// TIA Portal project "997CS100_KKD" (V16)

(* hardware
DEVICE "S71500/ET200MP station_1"  S7-1500 station
   slot 0: "-N01.01.00"  Rack  6ES7 590-1***0-0AA0
   slot 1: "997CS100"  CPU 1515-2 PN  6ES7 515-2AM02-0AB0  V2.8
      slot 3: "CPU display_1"  6ES7591-1BA00-0AA0
      slot 32768: "IO"  X1
      slot 33024: "PROFINET interface_1"  X2
      slot 34817: "Virtual CP interface port_1"  Virtual CP interface port  Virtual CP interface port
DEVICE "Station ET 200SP_7"  ET 200SP-Station
   slot 0: "Châssis_0"  6ES5 710-8MAx1
   slot 0: "PMC"  IM 155-6 PN ST  6ES7 155-6AU01-0BN0  V4.1
   slot 1: "501DI1"  DI 16x24VDC ST  6ES7 131-6BH01-0BA0  V0.0
      slot 1: "501DI1"  DI 16x24VDC ST
   slot 2: "501DI2"  DI 16x24VDC ST  6ES7 131-6BH01-0BA0  V0.0
      slot 1: "501DI2"  DI 16x24VDC ST
   slot 3: "501DI3"  DI 16x24VDC ST  6ES7 131-6BH01-0BA0  V0.0
      slot 1: "501DI3"  DI 16x24VDC ST
   slot 4: "501DI4"  DI 16x24VDC ST  6ES7 131-6BH01-0BA0  V0.0
      slot 1: "501DI4"  DI 16x24VDC ST
   slot 5: "501DI5"  DI 16x24VDC ST  6ES7 131-6BH01-0BA0  V0.0
      slot 1: "501DI5"  DI 16x24VDC ST
   slot 6: "502DO1"  RQ 4x120VDC/230VAC/5A NO ST  6ES7 132-6HD01-0BB1  V0.0
      slot 1: "502DO1"  RQ 4x120VDC/230VAC/5A NO ST
   slot 7: "502DO2"  RQ 4x120VDC/230VAC/5A NO ST  6ES7 132-6HD01-0BB1  V0.0
      slot 1: "502DO2"  RQ 4x120VDC/230VAC/5A NO ST
   slot 8: "502DO3"  RQ 4x120VDC/230VAC/5A NO ST  6ES7 132-6HD01-0BB1  V0.0
      slot 1: "502DO3"  RQ 4x120VDC/230VAC/5A NO ST
   slot 9: "502DO4"  RQ 4x120VDC/230VAC/5A NO ST  6ES7 132-6HD01-0BB1  V0.0
      slot 1: "502DO4"  RQ 4x120VDC/230VAC/5A NO ST
   slot 10: "502AI1"  AI 4xI 2-,4-wire ST  6ES7 134-6GD01-0BA1  V2.0
      slot 1: "502AI1"  AI 4xI 2-,4-wire ST
   slot 11: "502AI2"  AI 4xI 2-,4-wire ST  6ES7 134-6GD01-0BA1  V2.0
      slot 1: "502AI2"  AI 4xI 2-,4-wire ST
   slot 12: "502AI3"  AI 8xI 2-,4-wire BA  6ES7 134-6GF00-0AA1  V1.0
      slot 1: "502AI3"  AI 8xI 2-,4-wire BA
   slot 13: "300DI1"  DI 16x24VDC ST  6ES7 131-6BH01-0BA0  V0.0
      slot 1: "300DI1"  DI 16x24VDC ST
   slot 14: "300DI2"  DI 16x24VDC ST  6ES7 131-6BH01-0BA0  V0.0
      slot 1: "300DI2"  DI 16x24VDC ST
   slot 15: "300DI3"  DI 16x24VDC ST  6ES7 131-6BH01-0BA0  V0.0
      slot 1: "300DI3"  DI 16x24VDC ST
   slot 16: "300DO1"  DQ 16x24VDC/0.5A ST  6ES7 132-6BH01-0BA0  V0.0
      slot 1: "300DO1"  DQ 16x24VDC/0.5A ST
   slot 17: "Module serveur_1"  Module serveur  6ES7 193-6PA00-0AA0  V1.0
      slot 1: "Module serveur_1"  Module serveur
   slot 127: "Adaptateur de bus PROFINET CU"  PROFINET Interface  6ES7 193-6AR00-0AA0  V0.0
      slot 1: "Port_1"  6ES7 193-6AR00-0AA0  V0.0
      slot 2: "Port_2"  6ES7 193-6AR00-0AA0  V0.0
DEVICE "GSD device_2"  GSD.Device.PN
   slot 0: "Rack"  Rack  V1.0
   slot 0: "CV180_VFD"  INVT Profinet Adapter V1.0  1234567  V13.00.00
      slot 0: "INVT Profinet Adapter board V1.0"  INVT Profinet Adapter board V1.0
      slot 1: "PN-IO"  PN-IO
         slot 1: "Port 1 - RJ45"  Port 1 - RJ45
         slot 2: "Port 2 - RJ45"  Port 2 - RJ45
   slot 1: "32 Byte IN/OUT_1"  32 Byte IN/OUT  1.0
      slot 0: "32 Byte IN/OUT"  32 Byte IN/OUT
DEVICE "2010CV300U01_INVT"  GSD.Device.PN
   slot 0: "Rack"  Rack  V1.0
   slot 0: "2010CV300U01_INVT"  INVT Profinet Adapter V1.0  1234567  V13.00.00
      slot 0: "INVT Profinet Adapter board V1.0"  INVT Profinet Adapter board V1.0
      slot 1: "PN-IO"  PN-IO
         slot 1: "Port 1 - RJ45"  Port 1 - RJ45
         slot 2: "Port 2 - RJ45"  Port 2 - RJ45
   slot 1: "32 Byte IN/OUT_1"  32 Byte IN/OUT  1.0
      slot 0: "32 Byte IN/OUT"  32 Byte IN/OUT
DEVICE "Control device Station"  SIMOCODE pro
   slot 0: "Rack"  Rail
   slot 0: "2010cv120m01"  SIMOCODE pro V PN  3UF7 011-1A*00-0  V2.1
      slot 1: "Control device IO_1"  3UF7 011-1A*00-0
   slot 101: "IM 2.4 - 25A"  Current measuring module 2.4..25A  3UF7 101-1*A00-0
DEVICE "ET 200SP station_1"  ET 200SP-Station
   slot 0: "-N02.01.00"  Rack  6ES5 710-8MAx1
   slot 0: "993CS110A01"  IM 155-6 PN/2 HF  6ES7 155-6AU01-0CN0  V4.2
   slot 1: "-N02.01.01"  DI 16x24VDC ST  6ES7 131-6BH01-0BA0  V0.0
      slot 1: "-N02.01.01"  DI 16x24VDC ST
   slot 2: "-N02.01.02"  AI 8xI 2-,4-wire BA  6ES7 134-6GF00-0AA1  V1.0
      slot 1: "-N02.01.02"  AI 8xI 2-,4-wire BA
   slot 3: "-N02.01.03"  AQ 4xU/I ST  6ES7 135-6HD00-0BA1  V1.1
      slot 1: "-N02.01.03"  AQ 4xU/I ST
   slot 4: "-N02.01.04"  DI 16x24VDC ST  6ES7 131-6BH01-0BA0  V0.0
      slot 1: "-N02.01.04"  DI 16x24VDC ST
   slot 5: "-N02.01.05"  DI 16x24VDC ST  6ES7 131-6BH01-0BA0  V0.0
      slot 1: "-N02.01.05"  DI 16x24VDC ST
   slot 6: "-N02.01.06"  DI 16x24VDC ST  6ES7 131-6BH01-0BA0  V0.0
      slot 1: "-N02.01.06"  DI 16x24VDC ST
   slot 7: "-N02.01.07"  DQ 16x24VDC/0.5A ST  6ES7 132-6BH01-0BA0  V0.0
      slot 1: "-N02.01.07"  DQ 16x24VDC/0.5A ST
   slot 8: "-N02.01.08"  DQ 16x24VDC/0.5A ST  6ES7 132-6BH01-0BA0  V0.0
      slot 1: "-N02.01.08"  DQ 16x24VDC/0.5A ST
   slot 9: "-N02.01.09"  DQ 16x24VDC/0.5A ST  6ES7 132-6BH01-0BA0  V0.0
      slot 1: "-N02.01.09"  DQ 16x24VDC/0.5A ST
   slot 10: "Server module_1"  Server module  6ES7 193-6PA00-0AA0  V1.1
      slot 1: "Server module_1"  Server module
   slot 127: "BA 2xRJ45"  BA 2xRJ45  6ES7 193-6AR00-0AA0  V0.0
      slot 1: "Port_1"  X1 P1 R  6ES7 193-6AR00-0AA0  V0.0
      slot 2: "Port_2"  X1 P2 R  6ES7 193-6AR00-0AA0  V0.0
DEVICE "997spareABB1"  GSD.Device.PN
   slot 0: "Rack"  Rack  V1.0
   slot 0: "997spareABB1"  FENA-21  6438177287452  V3.2.0
      slot 0: "FENA-21"  FENA-21
      slot 1: "997spareABB1"  Interface
         slot 1: "Port 1"  Port 1
         slot 2: "Port 2"  Port 2
   slot 1: "PPO Type 7_1"  PPO Type 7  V3.2.0
      slot 0: "PPO7 Data Object"  PPO7 Data Object
DEVICE "2015PU040U01"  GSD.Device.PN
   slot 0: "Rack"  Rack  V1.0
   slot 0: "2015PU040U01"  FENA-21  6438177287452  V3.2.0
      slot 0: "FENA-21"  FENA-21
      slot 1: "Interface"  Interface
         slot 1: "Port 1"  Port 1
         slot 2: "Port 2"  Port 2
   slot 1: "PPO Type 7_1"  PPO Type 7  V3.2.0
      slot 0: "PPO7 Data Object"  PPO7 Data Object
DEVICE "2015PU027U01"  GSD.Device.PN
   slot 0: "Rack"  Rack  V1.0
   slot 0: "2015PU027U01"  INVT Profinet Adapter V1.0  1234567  V13.00.00
      slot 0: "INVT Profinet Adapter board V1.0"  INVT Profinet Adapter board V1.0
      slot 1: "PN-IO"  PN-IO
         slot 1: "Port 1 - RJ45"  Port 1 - RJ45
         slot 2: "Port 2 - RJ45"  Port 2 - RJ45
   slot 1: "32 Byte IN/OUT_1"  32 Byte IN/OUT  1.0
      slot 0: "32 Byte IN/OUT"  32 Byte IN/OUT
DEVICE "2015PU028U01"  GSD.Device.PN
   slot 0: "Rack"  Rack  V1.0
   slot 0: "2015PU028U01"  INVT Profinet Adapter V1.0  1234567  V13.00.00
      slot 0: "INVT Profinet Adapter board V1.0"  INVT Profinet Adapter board V1.0
      slot 1: "PN-IO"  PN-IO
         slot 1: "Port 1 - RJ45"  Port 1 - RJ45
         slot 2: "Port 2 - RJ45"  Port 2 - RJ45
   slot 1: "32 Byte IN/OUT_1"  32 Byte IN/OUT  1.0
      slot 0: "32 Byte IN/OUT"  32 Byte IN/OUT
DEVICE "2015PU035U01"  GSD.Device.PN
   slot 0: "Rack"  Rack  V1.0
   slot 0: "2015PU035U01"  INVT Profinet Adapter V1.0  1234567  V13.00.00
      slot 0: "INVT Profinet Adapter board V1.0"  INVT Profinet Adapter board V1.0
      slot 1: "PN-IO"  PN-IO
         slot 1: "Port 1 - RJ45"  Port 1 - RJ45
         slot 2: "Port 2 - RJ45"  Port 2 - RJ45
   slot 1: "32 Byte IN/OUT_1"  32 Byte IN/OUT  1.0
      slot 0: "32 Byte IN/OUT"  32 Byte IN/OUT
DEVICE "2015PU042M01"  SIMOCODE pro
   slot 0: "UR"  Rail
   slot 0: "2015PU042M01"  SIMOCODE pro V PN GP  3UF7 011-1A*00-1  V2.1
      slot 1: "SIMOCODE"  3UF7 011-1A*00-1
   slot 10: "OP"  Operator Panel Titangrey  3UF7 200-1AA01-0
   slot 101: "IM 10-100A"  Current measuring module 10..100A  3UF7 102-1*A00-0
DEVICE "GSD device_3"  GSD.Device.PN
   slot 0: "Rack"  Rack  V1.0
   slot 0: "BF110_VFD"  ATV930  ATV930
      slot 0: "ATV930"  ATV930
      slot 1: "Interface"  Interface
         slot 1: "Port 1"  Port 1
         slot 2: "Port 2"  Port 2
   slot 1: "Telegram 107 (4PKW/16PZD)"  Telegram 107 (4PKW/16PZD)
      slot 0: "Telegram 107"  Telegram 107
DEVICE "GSD device_4"  GSD.Device.PN
   slot 0: "Rack"  Rack  V1.0
   slot 0: "SC130_VFD"  ATV930  ATV930
      slot 0: "ATV930"  ATV930
      slot 1: "Interface"  Interface
         slot 1: "Port 1"  Port 1
         slot 2: "Port 2"  Port 2
   slot 1: "Telegram 107 (4PKW/16PZD)"  Telegram 107 (4PKW/16PZD)
      slot 0: "Telegram 107"  Telegram 107
DEVICE "2010LV100P01"  GSD.Device.PN
   slot 0: "UR"  Rack  V1.0
   slot 0: "2010LV100P01"  PAC3220
      slot 0: "PAC3220"  PAC3220
      slot 1: "2010LV100P01"  PN-IO
         slot 1: "Port 1"  Port 1
         slot 2: "Port 2"  Port 2
   slot 1: "Digital Inputs Status"  Digital Inputs Status
      slot 0: "Digital Inputs Status"  Digital Inputs Status
   slot 2: "Voltage L1-L2"  Voltage L1-L2
      slot 0: "Voltage L1-L2"  Voltage L1-L2
   slot 3: "Voltage L2-L3"  Voltage L2-L3
      slot 0: "Voltage L2-L3"  Voltage L2-L3
   slot 4: "Voltage L3-L1"  Voltage L3-L1
      slot 0: "Voltage L3-L1"  Voltage L3-L1
   slot 5: "Current L1"  Current L1
      slot 0: "Current L1"  Current L1
   slot 6: "Current L2"  Current L2
      slot 0: "Current L2"  Current L2
   slot 7: "Current L3"  Current L3
      slot 0: "Current L3"  Current L3
   slot 8: "Line Frequency"  Line Frequency
      slot 0: "Line Frequency"  Line Frequency
   slot 9: "Total Apparent Power"  Total Apparent Power
      slot 0: "Total Apparent Power"  Total Apparent Power
   slot 10: "Total Active Power"  Total Active Power
      slot 0: "Total Active Power"  Total Active Power
   slot 11: "Total Reac Power"  Total Reac Power
      slot 0: "Total Reac Power"  Total Reac Power
   slot 12: "Total Power Factor"  Total Power Factor
      slot 0: "Total Power Factor"  Total Power Factor
   slot 13: "Act Energy Imp Tar 1(F)"  Act Energy Imp Tar 1(F)
      slot 0: "Act Energy Imp Tar 1(F)"  Act Energy Imp Tar 1(F)
   slot 14: "Reac En Imp Tar 1 (F)"  Reac En Imp Tar 1 (F)
      slot 0: "Reac En Imp Tar 1 (F)"  Reac En Imp Tar 1 (F)
   slot 15: "App Energy Tariff 1 (F)"  App Energy Tariff 1 (F)
      slot 0: "App Energy Tariff 1 (F)"  App Energy Tariff 1 (F)
DEVICE "Control device Station_1"  SIMOCODE pro
   slot 0: "Rack"  Rail
   slot 0: "2010SJ950M01"  SIMOCODE pro V PN  3UF7 011-1A*00-0  V2.1
      slot 1: "Control device IO_1"  3UF7 011-1A*00-0
   slot 10: "OP"  Operator Panel Titangrey  3UF7 200-1AA01-0
   slot 101: "IM 10 - 100A"  Current measuring module 10..100A  3UF7 102-1*A00-0
DEVICE "997spareSimocode01"  SIMOCODE pro
   slot 0: "Rack"  Rail
   slot 0: "997spareSimocode01"  SIMOCODE pro V PN GP  3UF7 011-1A*00-1  V2.1
      slot 1: "Control device IO_1"  3UF7 011-1A*00-1
   slot 10: "OP"  Operator Panel Titangrey  3UF7 200-1AA01-0
   slot 101: "IM 10 - 100A"  Current measuring module 10..100A  3UF7 102-1*A00-0
DEVICE "2015PU041M01"  SIMOCODE pro
   slot 0: "Rack"  Rail
   slot 0: "2015PU041M01"  SIMOCODE pro V PN  3UF7 011-1A*00-0  V2.1
      slot 1: "Control device IO_1"  3UF7 011-1A*00-0
   slot 10: "OP"  Operator Panel Titangrey  3UF7 200-1AA01-0
   slot 101: "IM 10 - 100A"  Current measuring module 10..100A  3UF7 102-1*A00-0
DEVICE "997spareSimocode02"  SIMOCODE pro
   slot 0: "Rack"  Rail
   slot 0: "997spareSimocode02"  SIMOCODE pro V PN GP  3UF7 011-1A*00-1  V2.1
      slot 1: "Control device IO_1"  3UF7 011-1A*00-1
   slot 10: "OP"  Operator Panel Titangrey  3UF7 200-1AA01-0
   slot 101: "IM 10 - 100A"  Current measuring module 10..100A  3UF7 102-1*A00-0
DEVICE "997spareSimocode03"  SIMOCODE pro
   slot 0: "Rack"  Rail
   slot 0: "997spareSimocode03"  SIMOCODE pro V PN GP  3UF7 011-1A*00-1  V2.1
      slot 1: "Control device IO_1"  3UF7 011-1A*00-1
   slot 10: "OP"  Operator Panel Titangrey  3UF7 200-1AA01-0
   slot 101: "IM 10 - 100A"  Current measuring module 10..100A  3UF7 102-1*A00-0
DEVICE "997spareSimocode04"  SIMOCODE pro
   slot 0: "Rack"  Rail
   slot 0: "997spareSimocode04"  SIMOCODE pro V PN GP  3UF7 011-1A*00-1  V2.1
      slot 1: "Control device IO_1"  3UF7 011-1A*00-1
   slot 10: "OP"  Operator Panel Titangrey  3UF7 200-1AA01-0
   slot 101: "IM 10 - 100A"  Current measuring module 10..100A  3UF7 102-1*A00-0
DEVICE "997spareSimocode05"  SIMOCODE pro
   slot 0: "Rack"  Rail
   slot 0: "997spareSimocode05"  SIMOCODE pro V PN GP  3UF7 011-1A*00-1  V2.1
      slot 1: "Control device IO_1"  3UF7 011-1A*00-1
   slot 10: "OP"  Operator Panel Titangrey  3UF7 200-1AA01-0
   slot 101: "IM 10 - 100A"  Current measuring module 10..100A  3UF7 102-1*A00-0
DEVICE "997spareINVT02"  GSD.Device.PN
   slot 0: "Rack"  Rack  V1.0
   slot 0: "997spareINVT02"  INVT Profinet Adapter V1.0  1234567  V13.00.00
      slot 0: "INVT Profinet Adapter board V1.0"  INVT Profinet Adapter board V1.0
      slot 1: "997spareINVT02"  PN-IO
         slot 1: "Port 1 - RJ45"  Port 1 - RJ45
         slot 2: "Port 2 - RJ45"  Port 2 - RJ45
   slot 1: "32 Byte IN/OUT_1"  32 Byte IN/OUT  1.0
      slot 0: "32 Byte IN/OUT"  32 Byte IN/OUT
DEVICE "997spareINVT03"  GSD.Device.PN
   slot 0: "Rack"  Rack  V1.0
   slot 0: "997spareINVT03"  INVT Profinet Adapter V1.0  1234567  V13.00.00
      slot 0: "INVT Profinet Adapter board V1.0"  INVT Profinet Adapter board V1.0
      slot 1: "997spareINVT03"  PN-IO
         slot 1: "Port 1 - RJ45"  Port 1 - RJ45
         slot 2: "Port 2 - RJ45"  Port 2 - RJ45
   slot 1: "32 Byte IN/OUT_1"  32 Byte IN/OUT  1.0
      slot 0: "32 Byte IN/OUT"  32 Byte IN/OUT
DEVICE "997spareINVT04"  GSD.Device.PN
   slot 0: "Rack"  Rack  V1.0
   slot 0: "997spareINVT04"  INVT Profinet Adapter V1.0  1234567  V13.00.00
      slot 0: "INVT Profinet Adapter board V1.0"  INVT Profinet Adapter board V1.0
      slot 1: "997spareINVT04"  PN-IO
         slot 1: "Port 1 - RJ45"  Port 1 - RJ45
         slot 2: "Port 2 - RJ45"  Port 2 - RJ45
   slot 1: "32 Byte IN/OUT_1"  32 Byte IN/OUT  1.0
      slot 0: "32 Byte IN/OUT"  32 Byte IN/OUT
DEVICE "997spareINVT05"  GSD.Device.PN
   slot 0: "Rack"  Rack  V1.0
   slot 0: "997spareINVT05"  INVT Profinet Adapter V1.0  1234567  V13.00.00
      slot 0: "INVT Profinet Adapter board V1.0"  INVT Profinet Adapter board V1.0
      slot 1: "997spareINVT05"  PN-IO
         slot 1: "Port 1 - RJ45"  Port 1 - RJ45
         slot 2: "Port 2 - RJ45"  Port 2 - RJ45
   slot 1: "32 Byte IN/OUT_1"  32 Byte IN/OUT  1.0
      slot 0: "32 Byte IN/OUT"  32 Byte IN/OUT
DEVICE "997spareABB2"  GSD.Device.PN
   slot 0: "Rack"  Rack  V1.0
   slot 0: "997spareABB2"  FENA-21  6438177287452  V3.2.0
      slot 0: "FENA-21"  FENA-21
      slot 1: "997spareABB2"  Interface
         slot 1: "Port 1"  Port 1
         slot 2: "Port 2"  Port 2
   slot 1: "PPO Type 7_1"  PPO Type 7  V3.2.0
      slot 0: "PPO7 Data Object"  PPO7 Data Object
DEVICE "997spareABB3"  GSD.Device.PN
   slot 0: "Rack"  Rack  V1.0
   slot 0: "997spareABB3"  FENA-21  6438177287452  V3.2.0
      slot 0: "FENA-21"  FENA-21
      slot 1: "997spareABB3"  Interface
         slot 1: "Port 1"  Port 1
         slot 2: "Port 2"  Port 2
   slot 1: "PPO Type 7_1"  PPO Type 7  V3.2.0
      slot 0: "PPO7 Data Object"  PPO7 Data Object
DEVICE "997spareABB4"  GSD.Device.PN
   slot 0: "Rack"  Rack  V1.0
   slot 0: "997spareABB4"  FENA-21  6438177287452  V3.2.0
      slot 0: "FENA-21"  FENA-21
      slot 1: "997spareABB5"  Interface
         slot 1: "Port 1"  Port 1
         slot 2: "Port 2"  Port 2
   slot 1: "PPO Type 7_1"  PPO Type 7  V3.2.0
      slot 0: "PPO7 Data Object"  PPO7 Data Object
DEVICE "997spareABB5"  GSD.Device.PN
   slot 0: "Rack"  Rack  V1.0
   slot 0: "997spareABB5"  FENA-21  6438177287452  V3.2.0
      slot 0: "FENA-21"  FENA-21
      slot 1: "997spareABB5"  Interface
         slot 1: "Port 1"  Port 1
         slot 2: "Port 2"  Port 2
   slot 1: "PPO Type 7_1"  PPO Type 7  V3.2.0
      slot 0: "PPO7 Data Object"  PPO7 Data Object
DEVICE "2010CV300U01_ABB"  GSD.Device.PN
   slot 0: "Rack"  Rack  V1.0
   slot 0: "2010CV300U01_ABB"  FENA-21  6438177287452  V3.2.0
      slot 0: "FENA-21"  FENA-21
      slot 1: "Interface"  Interface
         slot 1: "Port 1"  Port 1
         slot 2: "Port 2"  Port 2
   slot 1: "PPO Type 7_1"  PPO Type 7  V3.2.0
      slot 0: "PPO7 Data Object"  PPO7 Data Object
*)

// ===== PLC "997CS100"  CPU 1515-2 PN =====

VAR_GLOBAL   // PLC tag table "Default tag table"
   "Clock_0.1Hz_tmp" AT %M3.1 : Bool;
   "Clock_0.1Hz" AT %M3.0 : Bool;
   "_997MS100_O1" AT %M1116.0 : Bool;
   "_997MS100_New_Shift_Pulse" AT %M1116.1 : Bool;
   "_997MS100_O2" AT %M1116.2 : Bool;
   "_997MS100_New_Day_Pulse" AT %M1116.3 : Bool;
   "System_Byte" AT %MB1 : Byte;
   "FirstScan" AT %M1.0 : Bool;
   "DiagStatusUpdate" AT %M1.1 : Bool;
   "Clock_Byte" AT %MB2 : Byte;
   "Clock_10Hz" AT %M2.0 : Bool;
   "Clock_5Hz" AT %M2.1 : Bool;
   "Clock_2.5Hz" AT %M2.2 : Bool;
   "Clock_2Hz" AT %M2.3 : Bool;
   "Clock_1.25Hz" AT %M2.4 : Bool;
   "Clock_1Hz" AT %M2.5 : Bool;
   "Clock_0.625Hz" AT %M2.6 : Bool;
   "Clock_0.5Hz" AT %M2.7 : Bool;
   "_2010LV100Q02E41" AT %I12.0 : Bool;   // Power Supply OK
   "_2010LV100F31E41" AT %I12.1 : Bool;   // Power Supply OK
   "_2010LV100F41E41" AT %I12.3 : Bool;   // Power Supply OK
   "_2010LV100C01U41" AT %I12.4 : Bool;   // Capacitor General Fault
   "SPARE_DI12_6" AT %I12.6 : Bool;   // Spare
   "_2010LCP300U01SSW02" AT %I12.7 : Bool;   // Button "ES" near the driveshaft is pressed
   "_2010LCP300U01SSW03" AT %I13.0 : Bool;   // Button "ES" near the non-drive shaft is pressed
   "_2010LCP300U01LOC" AT %I13.1 : Bool;
   "_2010LCP300U01AMS" AT %I13.2 : Bool;   // Control mode "REMOTE"
   "_2010LCP300U01REP" AT %I13.3 : Bool;   // Control mode "REPAIR"
   "_2010LCP300U01STP" AT %I13.4 : Bool;   // The "STOP" command
   "_2010LCP300U01STR" AT %I13.5 : Bool;   // The "START" command
   "_2010LCP300U01RES" AT %I13.6 : Bool;   // Resetting an accident
   "_2010CV300D21Z41" AT %I14.0 : Bool;   // Local Start
   "_2010CV300D22Z41" AT %I14.1 : Bool;   // Local Stop
   "_2010CV300D02S41" AT %I14.2 : Bool;   // Датчик скорости на 2м барабане
   "_2010CR150A01T01" AT %IW272 : Int;   // темп. подшипника левый неподвижный
   "_2010CR150A01T02" AT %IW274 : Int;   // темп. подшипника правый неподвижный
   "_2010CR150A01T03" AT %IW276 : Int;   // темп. подшипника правый подвижный
   "_2010CR150A01T04" AT %IW278 : Int;   // темп. подшипника левый подвижный
   "Conv120.Simocode.SW" AT %IW570 : Int;   // Conv120 Simocode Status Word
   "Conv120.Simocode.AI" AT %IW572 : Int;   // Conv120 Simocode Analog Reading (%ls)
   "_2010CV300N01T01" AT %IW280 : Int;   // Reducer Temp
   "_2010CV180U01C53" AT %M1001.0 : Bool;   // Local Stop
   "_2010CV180U01C51" AT %M1001.1 : Bool;   // Local Start
   "_2010CV180U01C73" AT %M1001.2 : Bool;   // Unbalance
   "_2010CV180U01C42" AT %M1001.3 : Bool;   // Drive / MCC Ready
   "_2010CV180U01C71" AT %M1001.4 : Bool;   // Motor Stalled
   "_2010CV180U01C45" AT %M1001.5 : Bool;   // Drawer Test Pos.
   "_2010CV180U01U41" AT %M1001.6 : Bool;   // General Fault
   "_2010CV180U01C44" AT %M1001.7 : Bool;   // Overload
   "_2010CV180U01C46" AT %M1002.0 : Bool;   // Bus Fault
   "_2010CV180U01C47" AT %M1002.1 : Bool;   // Drawer Oper. Pos.
   "_2010CV180U01C72" AT %M1002.2 : Bool;   // Earth Fault
   "_2010CV180U01C74" AT %M1002.3 : Bool;   // Reset Ack.
   "_2010CV180U01U42" AT %M1002.4 : Bool;   // General Warning
   "_2010CV180U01C56" AT %M1002.5 : Bool;   // Safety Switch
   "_2010CV180U01C61" AT %M1002.6 : Bool;   // Return
   "_2010CV180U01I01" AT %MD3038 : Real;   // Current
   "_2010CV180U01J01" AT %MD3042 : Real;   // Power
   "_2010CV180U01S01" AT %MD3046 : Real;   // Speed
   "_2010CV180U01S11" AT %MD3050 : Real;   // Speed Setpoint
   "_2010CV120M01I01" AT %MD3054 : Real;   // Current
   "_2010CV120M01J01" AT %MD3058 : Real;   // Power
   "_2010CV120M01S01" AT %MD3062 : Real;   // Speed
   "_2010BF110U01J01" AT %MD3066 : Real;   // Speed Setpoint
   "_2010CV120M01C53" AT %M1005.0 : Bool;   // Local Stop
   "_2010CV120M01C51" AT %M1005.1 : Bool;   // Local Start
   "_2010CV120M01C73" AT %M1005.2 : Bool;   // Unbalance
   "_2010CV120M01C42" AT %M1005.3 : Bool;   // Drive / MCC Ready
   "_2010CV120M01C71" AT %M1005.4 : Bool;   // Motor Stalled
   "_2010CV120M01C45" AT %M1005.5 : Bool;   // Drawer Test Pos.
   "_2010CV120M01U41" AT %M1005.6 : Bool;   // General Fault
   "_2010CV120M01C44" AT %M1005.7 : Bool;   // Overload
   "_2010CV120M01C46" AT %M1006.0 : Bool;   // Bus Fault
   "_2010CV120M01C47" AT %M1006.1 : Bool;   // Drawer Oper. Pos.
   "_2010CV120M01C72" AT %M1006.2 : Bool;   // Earth Fault
   "_2010CV120M01C74" AT %M1006.3 : Bool;   // Reset Ack.
   "_2010CV120M01U42" AT %M1006.4 : Bool;   // General Warning
   "_2010CV120M01C56" AT %M1006.5 : Bool;   // Safety Switch
   "_2010CV120M01C61" AT %M1006.6 : Bool;   // Return
   "_2010CV190M01C53" AT %M1007.0 : Bool;   // Local Stop
   "_2010OB190M01C51" AT %M1007.1 : Bool;   // Local Start
   "_2010OB190M01C73" AT %M1007.2 : Bool;   // Unbalance
   "_2010OB190M01C42" AT %M1007.3 : Bool;   // Drive / MCC Ready
   "_2010OB190M01C71" AT %M1007.4 : Bool;   // Motor Stalled
   "_2010OB190M01C45" AT %M1007.5 : Bool;   // Drawer Test Pos.
   "_2010OB190M01U41" AT %M1007.6 : Bool;   // General Fault
   "_2010OB190M01C44" AT %M1007.7 : Bool;   // Overload
   "_2010OB190M01C46" AT %M1008.0 : Bool;   // Bus Fault
   "_2010OB190M01C47" AT %M1008.1 : Bool;   // Drawer Oper. Pos.
   "_2010OB190M01C72" AT %M1008.2 : Bool;   // Earth Fault
   "_2010OB190M01C74" AT %M1008.3 : Bool;   // Reset Ack.
   "_2010OB190M01U42" AT %M1008.4 : Bool;   // General Warning
   "_2010OB190M01C56" AT %M1008.5 : Bool;   // Safety Switch
   "_2010OB190M01C61" AT %M1008.6 : Bool;   // Return
   "_2010BF110U01C53" AT %M1010.0 : Bool;   // Local Stop
   "_2010BF110U01C51" AT %M1010.1 : Bool;   // Local Start
   "_2010BF110U01C73" AT %M1010.2 : Bool;   // Unbalance
   "_2010BF110U01C42" AT %M1010.3 : Bool;   // Drive / MCC Ready
   "_2010BF110U01C71" AT %M1010.4 : Bool;   // Motor Stalled
   "_2010BF110U01C45" AT %M1010.5 : Bool;   // Drawer Test Pos.
   "_2010BF110U01U41" AT %M1010.6 : Bool;   // General Fault
   "_2010BF110U01C44" AT %M1010.7 : Bool;   // Overload
   "_2010BF110U01C46" AT %M1011.0 : Bool;   // Bus Fault
   "_2010BF110U01C47" AT %M1011.1 : Bool;   // Drawer Oper. Pos.
   "_2010BF110U01C72" AT %M1011.2 : Bool;   // Earth Fault
   "_2010BF110U01C74" AT %M1011.3 : Bool;   // Reset Ack.
   "_2010BF110U01U42" AT %M1011.4 : Bool;   // General Warning
   "_2010BF110U01C56" AT %M1011.5 : Bool;   // Safety Switch
   "_2010BF110U01C61" AT %M1011.6 : Bool;   // Return
   "_2010BF110U01S01" AT %MD3074 : Real;   // Speed
   "_2010BF110U01S11" AT %MD3078 : Real;   // Speed Setpoint
   "_2010BF110U01I01" AT %MD3070 : Real;   // Current
   "_2010SC130U01C53" AT %M1012.0 : Bool;   // Local Stop
   "_2010SC130U01C51" AT %M1012.1 : Bool;   // Local Start
   "_2010SC130U01C73" AT %M1012.2 : Bool;   // Unbalance
   "_2010SC130U01C42" AT %M1012.3 : Bool;   // Drive / MCC Ready
   "_2010SC130U01C71" AT %M1012.4 : Bool;   // Motor Stalled
   "_2010SC130U01C45" AT %M1012.5 : Bool;   // Drawer Test Pos.
   "_2010SC130U01U41" AT %M1012.6 : Bool;   // General Fault
   "_2010SC130U01C44" AT %M1012.7 : Bool;   // Overload
   "_2010SC130U01C46" AT %M1013.0 : Bool;   // Bus Fault
   "_2010SC130U01C47" AT %M1013.1 : Bool;   // Drawer Oper. Pos.
   "_2010SC130U01C72" AT %M1013.2 : Bool;   // Earth Fault
   "_2010SC130U01C74" AT %M1013.3 : Bool;   // Reset Ack.
   "_2010SC130U01U42" AT %M1013.4 : Bool;   // General Warning
   "_2010SC130U01C56" AT %M1013.5 : Bool;   // Safety Switch
   "_2010SC130U01C61" AT %M1013.6 : Bool;   // Return
   "_2010SC130U01I01" AT %MD3082 : Real;   // Current
   "_2010SC130U01S01" AT %MD3086 : Real;   // Speed
   "_2010SC130U01S11" AT %MD3090 : Real;   // Speed Setpoint
   "_2010SC130U01J01" AT %MD3094 : Real;   // Power
   "_2010CR150M01C53" AT %M1014.0 : Bool;   // Local Stop
   "_2010CR150M01C51" AT %M1014.1 : Bool;   // Local Start
   "_2010CR150M01C73" AT %M1014.2 : Bool;   // Unbalance
   "_2010CR150M01C42" AT %M1014.3 : Bool;   // Drive / MCC Ready
   "_2010CR150M01C71" AT %M1014.4 : Bool;   // Motor Stalled
   "_2010CR150M01C45" AT %M1014.5 : Bool;   // Drawer Test Pos.
   "_2010CR150M01U41" AT %M1014.6 : Bool;   // General Fault
   "_2010CR150M01C44" AT %M1014.7 : Bool;   // Overload
   "_2010CR150M01C46" AT %M1015.0 : Bool;   // Bus Fault
   "_2010CR150M01C47" AT %M1015.1 : Bool;   // Drawer Oper. Pos.
   "_2010CR150M01C72" AT %M1015.2 : Bool;   // Earth Fault
   "_2010CR150M01C74" AT %M1015.3 : Bool;   // Reset Ack.
   "_2010CR150M01U42" AT %M1015.4 : Bool;   // General Warning
   "_2010CR150M01C56" AT %M1015.5 : Bool;   // Safety Switch
   "_2010CR150M01C61" AT %M1015.6 : Bool;   // Return
   "_2010CV300ONS01" AT %M1016.0 : Bool;   // PulseOne
   "_2010SC130U01_MB_FRM_ERR" AT %M1013.7 : Bool;   // ModBus Comm Err
   "_2010BF110U01_MB_FRM_ERR" AT %M1011.7 : Bool;   // ModBus Comm Err
   "_2010SC130U01_new_spd" AT %M1016.1 : Bool;
   "_2010BF110U01_new_spd" AT %M1016.2 : Bool;
   "_2010SC130U01_SP_old" AT %MD3098 : Real;
   "_2010BF110U01_SP_old" AT %MD3102 : Real;
   "_2010CR150A01T05" AT %IW282 : Int;   // Темп. рядом с вибровозбудителем
   "_997CD100G03_start_warning" AT %M1016.3 : Bool;
   "100CV300H01C31" AT %Q10.0 : Bool;   // Command Light
   "100CV300H01C32" AT %Q10.1 : Bool;   // Command Horn
   "100CV300H02C31" AT %Q10.2 : Bool;   // Command Light
   "100CV300H02C32" AT %Q10.3 : Bool;   // Command Horn
   "100CV300H03C31" AT %Q10.4 : Bool;   // Command Light
   "100CV300H03C32" AT %Q10.5 : Bool;   // Command Horn
   "100CV300H04C31" AT %Q10.6 : Bool;   // Command Light
   "100CV300H04C32" AT %Q10.7 : Bool;   // Command Horn
   "100CV300H05C31" AT %Q11.0 : Bool;   // Command Light
   "100CV300U01RDY" AT %Q100.0 : Bool;   // Conveyor Ready
   "100CV300U01TRP" AT %Q100.1 : Bool;   // Conveyor Crash
   "100CV300U01SSW" AT %Q100.2 : Bool;   // Emergency stop
   "100CV300U01Z41" AT %Q100.3 : Bool;   // Fence open
   "100CV300U01RUN" AT %Q100.4 : Bool;   // WORK
   "997CD100G03ONS01" AT %M1016.5 : Bool;
   "997CD100G03ONS02" AT %M1016.6 : Bool;
   "997CD100G03ONS03" AT %M1016.7 : Bool;
   "997CD100G03ONS04" AT %M1017.0 : Bool;
   "997CD100G03ONS06" AT %M1017.1 : Bool;
   "997CD100G03ONS07" AT %M1017.2 : Bool;
   "997CD100G03ONS05" AT %M1017.3 : Bool;
   "_2010CV300U01MCC01" AT %M1018.0 : Bool;   // Power Supply Fault
   "_2010CV300U01SWW01" AT %M1018.1 : Bool;   // Seafety Fault
   "CV300_VFD_SB" AT %IB508 : Byte;
   "CV300VFD_Status" AT %IB59 : Byte;   // Spare
   "CV180_VFD_ SB" AT %IB540 : Byte;
   "CV180_VFD_ SB_Running_State" AT %IB541 : Byte;
   "CV300_VFD_ SB_IO" AT %IB525 : Byte;
   "CV180_VFD_ IO" AT %IB557 : Byte;
   "_2010SC130U01_mb_cmd_old" AT %MW3106 : Int;
   "_2010BF110U01_mb_cmd_old" AT %MW3108 : Int;
   "_2010SC130U01_wcmd" AT %M1017.4 : Bool;
   "_2010BF110U01_wcmd" AT %M1017.5 : Bool;
   "_2015PU027U01C42" AT %M1405.4 : Bool;   // Spare motor, Drive / MCC Ready
   "_2015PU027U01C44" AT %M1406.0 : Bool;   // Spare motor, Overload
   "_2015PU027U01C45" AT %M1405.6 : Bool;   // Spare motor, Drawer Test Pos.
   "_2015PU027U01C46" AT %M1406.1 : Bool;   // Spare motor, Bus Fault
   "_2015PU027U01C47" AT %M1406.2 : Bool;   // Spare motor, Drawer Oper. Pos.
   "_2015PU027U01C51" AT %M1405.1 : Bool;   // Spare motor, Local Start
   "_2015PU027U01C53" AT %M1405.0 : Bool;   // Spare motor, Local Stop
   "_2015PU027U01C56" AT %M1406.6 : Bool;   // Spare motor, Safety Switch
   "_2015PU027U01C61" AT %M1405.3 : Bool;   // Spare motor, Return
   "_2015PU027U01C71" AT %M1405.5 : Bool;   // Spare motor, Motor Stalled
   "_2015PU027U01C72" AT %M1406.3 : Bool;   // Spare motor, Earth Fault
   "_2015PU027U01C73" AT %M1405.2 : Bool;   // Spare motor, Unbalance
   "_2015PU027U01C74" AT %M1406.4 : Bool;   // Spare motor, Reset Ack.
   "_2015PU027U01I01" AT %MD4384 : Real;   // Spare Motor, Current
   "_2015PU027U01J01" AT %MD4388 : Real;   // Spare Motor, Power
   "_2015PU027U01S01" AT %MD4392 : Real;   // Spare Motor, Speed
   "_2015PU027U01U41" AT %M1405.7 : Bool;   // Spare motor, General Fault
   "_2015PU027U01U42" AT %M1406.5 : Bool;   // Spare motor, General Warning
   "_2015PU028U01C42" AT %M1407.4 : Bool;   // Spare motor, Drive / MCC Ready
   "_2015PU028U01C44" AT %M1408.0 : Bool;   // Spare motor, Overload
   "_2015PU028U01C45" AT %M1407.6 : Bool;   // Spare motor, Drawer Test Pos.
   "_2015PU028U01C46" AT %M1408.1 : Bool;   // Spare motor, Bus Fault
   "_2015PU028U01C47" AT %M1408.2 : Bool;   // Spare motor, Drawer Oper. Pos.
   "_2015PU028U01C51" AT %M1407.1 : Bool;   // Spare motor, Local Start
   "_2015PU028U01C53" AT %M1407.0 : Bool;   // Spare motor, Local Stop
   "_2015PU028U01C56" AT %M1408.6 : Bool;   // Spare motor, Safety Switch
   "_2015PU028U01C61" AT %M1407.3 : Bool;   // Spare motor, Return
   "_2015PU028U01C71" AT %M1407.5 : Bool;   // Spare motor, Motor Stalled
   "_2015PU028U01C72" AT %M1408.3 : Bool;   // Spare motor, Earth Fault
   "_2015PU028U01C73" AT %M1407.2 : Bool;   // Spare motor, Unbalance
   "_2015PU028U01C74" AT %M1408.4 : Bool;   // Spare motor, Reset Ack.
   "_2015PU028U01I01" AT %MD4400 : Real;   // Spare Motor, Current
   "_2015PU028U01J01" AT %MD4404 : Real;   // Spare Motor, Power
   "_2015PU028U01S01" AT %MD4408 : Real;   // Spare Motor, Speed
   "_2015PU028U01U41" AT %M1407.7 : Bool;   // Spare motor, General Fault
   "_2015PU028U01U42" AT %M1408.5 : Bool;   // Spare motor, General Warning
   "_2015PU035U01C42" AT %M1425.4 : Bool;
   "_2015PU035U01C44" AT %M1424.0 : Bool;
   "_2015PU035U01C45" AT %M1425.6 : Bool;
   "_2015PU035U01C46" AT %M1424.1 : Bool;
   "_2015PU035U01C47" AT %M1424.2 : Bool;
   "_2015PU035U01C51" AT %M1425.1 : Bool;
   "_2015PU035U01C53" AT %M1425.0 : Bool;
   "_2015PU035U01C56" AT %M1424.6 : Bool;
   "_2015PU035U01C61" AT %M1425.3 : Bool;
   "_2015PU035U01C71" AT %M1425.5 : Bool;
   "_2015PU035U01C72" AT %M1424.3 : Bool;
   "_2015PU035U01C73" AT %M1425.2 : Bool;
   "_2015PU035U01C74" AT %M1424.4 : Bool;
   "_2015PU035U01I01" AT %MD4556 : Real;
   "_2015PU035U01J01" AT %MD4560 : Real;
   "_2015PU035U01S01" AT %MD4564 : Real;
   "_2015PU035U01U41" AT %M1425.7 : Bool;
   "_2015PU035U01U42" AT %M1424.5 : Bool;
   "_2015PU040U01C42" AT %M1374.4 : Bool;   // Circulation Pump Crusher, Drive / MCC Ready
   "_2015PU040U01C44" AT %M1375.0 : Bool;   // Circulation Pump Crusher, Overload
   "_2015PU040U01C45" AT %M1374.6 : Bool;   // Circulation Pump Crusher, Drawer Test Pos.
   "_2015PU040U01C46" AT %M1375.1 : Bool;   // Circulation Pump Crusher, Bus Fault
   "_2015PU040U01C47" AT %M1375.2 : Bool;   // Circulation Pump Crusher, Drawer Oper. Pos.
   "_2015PU040U01C51" AT %M1374.1 : Bool;   // Circulation Pump Crusher, Local Start
   "_2015PU040U01C53" AT %M1374.0 : Bool;   // Circulation Pump Crusher, Local Stop
   "_2015PU040U01C56" AT %M1375.6 : Bool;   // Circulation Pump Crusher, Safety Switch
   "_2015PU040U01C61" AT %M1374.3 : Bool;   // Circulation Pump Crusher, Return
   "_2015PU040U01C71" AT %M1374.5 : Bool;   // Circulation Pump Crusher, Motor Stalled
   "_2015PU040U01C72" AT %M1375.3 : Bool;   // Circulation Pump Crusher, Earth Fault
   "_2015PU040U01C73" AT %M1374.2 : Bool;   // Circulation Pump Crusher, Unbalance
   "_2015PU040U01C74" AT %M1375.4 : Bool;   // Circulation Pump Crusher, Reset Ack.
   "_2015PU040U01I01" AT %MD4448 : Real;   // Spare Motor, Current
   "_2015PU040U01J01" AT %MD4452 : Real;   // Spare Motor, Power
   "_2015PU040U01S01" AT %MD4456 : Real;   // Spare Motor, Speed
   "_2015PU040U01S11" AT %MD4460 : Real;   // Spare Motor, Speed Setpoint
   "_2015PU040U01U41" AT %M1374.7 : Bool;   // Circulation Pump Crusher, General Fault
   "_2015PU040U01U42" AT %M1375.5 : Bool;   // Circulation Pump Crusher, General Warning
   "_2015PU041M01C42" AT %M1376.4 : Bool;   // Circulation Pump Crusher, Drive / MCC Ready
   "_2015PU041M01C44" AT %M1377.0 : Bool;   // Circulation Pump Crusher, Overload
   "_2015PU041M01C45" AT %M1376.6 : Bool;   // Circulation Pump Crusher, Drawer Test Pos.
   "_2015PU041U01C46" AT %M1377.1 : Bool;   // Circulation Pump Crusher, Bus Fault
   "_2015PU041M01C47" AT %M1377.2 : Bool;   // Circulation Pump Crusher, Drawer Oper. Pos.
   "_2015PU041M01C51" AT %M1376.1 : Bool;   // Circulation Pump Crusher, Local Start
   "_2015PU041M01C53" AT %M1376.0 : Bool;   // Circulation Pump Crusher, Local Stop
   "_2015PU041M01C56" AT %M1377.6 : Bool;   // Circulation Pump Crusher, Safety Switch
   "_2015PU041M01C61" AT %M1376.3 : Bool;   // Circulation Pump Crusher, Return
   "_2015PU041M01C71" AT %M1376.5 : Bool;   // Circulation Pump Crusher, Motor Stalled
   "_2015PU041M01C72" AT %M1377.3 : Bool;   // Circulation Pump Crusher, Earth Fault
   "_2015PU041M01C73" AT %M1376.2 : Bool;   // Circulation Pump Crusher, Unbalance
   "_2015PU041M01C74" AT %M1377.4 : Bool;   // Circulation Pump Crusher, Reset Ack.
   "_2015PU041M01I01" AT %MD4464 : Real;   // Spare Motor, Current
   "_2015PU041M01J01" AT %MD4468 : Real;   // Spare Motor, Power
   "_2015PU041U01S01" AT %MD4472 : Real;   // Spare Motor, Speed
   "_2015PU041U01S11" AT %MD4476 : Real;   // Spare Motor, Speed Setpoint
   "_2015PU041M01U41" AT %M1376.7 : Bool;   // Circulation Pump Crusher, General Fault
   "_2015PU041M01U42" AT %M1377.5 : Bool;   // Circulation Pump Crusher, General Warning
   "_2015PU042M01C44" AT %M1418.0 : Bool;   // Spare motor, Overload
   "_2015PU042M01C45" AT %M1417.6 : Bool;   // Spare motor, Drawer Test Pos.
   "_2015PU042M01C46" AT %M1418.1 : Bool;   // Spare motor, Bus Fault
   "_2015PU042M01C47" AT %M1418.2 : Bool;   // Spare motor, Drawer Oper. Pos.
   "_2015PU042M01C56" AT %M1418.6 : Bool;   // Spare motor, Safety Switch
   "_2015PU042M01C71" AT %M1417.5 : Bool;   // Spare motor, Motor Stalled
   "_2015PU042M01C72" AT %M1418.3 : Bool;   // Spare motor, Earth Fault
   "_2015PU042M01C74" AT %M1418.4 : Bool;   // Spare motor, Reset Ack.
   "_2015PU042M01I01" AT %MD4480 : Real;   // Glycol circulation pump, Current
   "_2015PU042M01J01" AT %MD4484 : Real;   // Glycol circulation pump, Power
   "_2015PU042M01S01" AT %MD4488 : Real;   // Glycol circulation pump, Speed
   "_2015PU042M01S11" AT %MD4492 : Real;   // Glycol circulation pump, Speed Setpoint
   "_2015PU042M01U41" AT %M1417.7 : Bool;   // Spare motor, General Fault
   "_2015PU042M01U42" AT %M1418.5 : Bool;   // Spare motor, General Warning
   "_2015PU042M01C53" AT %M1417.0 : Bool;   // Spare motor, Local Stop
   "_2015PU042M01C51" AT %M1417.1 : Bool;   // Spare motor, Local Start
   "_2015PU042M01C73" AT %M1417.2 : Bool;   // Spare motor, Unbalance
   "_2015PU042M01C61" AT %M1417.3 : Bool;   // Spare motor, Return
   "_2015PU042M01C42" AT %M1417.4 : Bool;   // Spare motor, Drive / MCC Ready
   "_2010BF110U01ONS01" AT %M1019.0 : Bool;
   "_2010BF110U01ONS02" AT %M1019.1 : Bool;
   "_2010CV300D19Z43" AT %I14.5 : Bool;   // Pull Rope Right Side Bottom
   "_2010CV300D20Z42" AT %I14.7 : Bool;   // Pull Rope Left Side Middle
   "_2010CV300D20Z41" AT %I14.6 : Bool;   // Pull Rope Left Side Top
   "_2010CV300D20Z43" AT %I15.0 : Bool;   // Pull Rope Left Side Bottom
   "_2010CV300D19Z41" AT %I14.3 : Bool;   // Pull Rope Right Side Top
   "_2010CV300D19Z42" AT %I14.4 : Bool;   // Pull Rope Right Side Middle
   "SPARE_DI12_2" AT %I12.2 : Bool;   // Spare
   "SPARE_DI13_7" AT %I13.7 : Bool;   // Spare
   "SPARE_DI15_1" AT %I15.1 : Bool;   // Spare
   "SPARE_DI15_2" AT %I15.2 : Bool;   // Spare
   "SPARE_DI15_3" AT %I15.3 : Bool;   // Spare
   "SPARE_DI15_4" AT %I15.4 : Bool;   // Spare
   "SPARE_DI15_5" AT %I15.5 : Bool;   // Spare
   "SPARE_DI15_6" AT %I15.6 : Bool;   // Spare
   "SPARE_DI15_7" AT %I15.7 : Bool;   // Spare
   "100CV300H05C32" AT %Q11.1 : Bool;   // Command Horn
   "SPARE_DO11_2" AT %Q11.2 : Bool;   // Spare
   "SPARE_DO11_3" AT %Q11.3 : Bool;   // Spare
   "SPARE_DO11_4" AT %Q11.4 : Bool;   // Spare
   "SPARE_DO11_5" AT %Q11.5 : Bool;   // Spare
   "SPARE_DO11_6" AT %Q11.6 : Bool;   // Spare
   "SPARE_DO11_7" AT %Q11.7 : Bool;   // Spare
   "_2010PMC01A01T01" AT %IW284 : Int;   // Температура в шкафу PMC
   "SPARE_AI286" AT %IW286 : Int;   // Spare
   "_MTR_SPAREC53" AT %M1020.0 : Bool;   // Local Stop
   "_MTR_SPAREC51" AT %M1020.1 : Bool;   // Local Start
   "_MTR_SPAREC73" AT %M1020.2 : Bool;   // Unbalance
   "_MTR_SPAREC42" AT %M1020.3 : Bool;   // Drive / MCC Ready
   "_MTR_SPAREC71" AT %M1020.4 : Bool;   // Motor Stalled
   "_MTR_SPAREC45" AT %M1020.5 : Bool;   // Drawer Test Pos.
   "_MTR_SPAREU41" AT %M1020.6 : Bool;   // General Fault
   "_MTR_SPAREC44" AT %M1020.7 : Bool;   // Overload
   "_MTR_SPAREC46" AT %M1021.0 : Bool;   // Bus Fault
   "_MTR_SPAREC47" AT %M1021.1 : Bool;   // Drawer Oper. Pos.
   "_MTR_SPAREC72" AT %M1021.2 : Bool;   // Earth Fault
   "_MTR_SPAREC74" AT %M1021.3 : Bool;   // Reset Ack.
   "_MTR_SPAREU42" AT %M1021.4 : Bool;   // General Warning
   "_MTR_SPAREC56" AT %M1021.5 : Bool;   // Safety Switch
   "_MTR_SPAREC61" AT %M1021.6 : Bool;   // Return
   "_MTR_SPARECI01" AT %MD4568 : Real;
   "_MTR_SPARECJ01" AT %MD4572 : Real;
   "_MTR_SPARECS01" AT %MD4576 : Real;
   "_2010LV100P01_App Energy Tariff 1 (F)" AT %ID6212 : Real;
   "Tag_1" AT %M1022.0 : Bool;
   "Tag_2" AT %M1022.1 : Bool;
   "Tag_3" AT %M1022.7 : Bool;
END_VAR

VAR_GLOBAL   // PLC tag table "STEP7 classic symbols"
   "AON_PROCESS1_BOOL" AT %M1000.5 : Bool;   // Logic Discuss With Process
   "AON_AFTERPLC_BOOL" AT %M1000.4 : Bool;   // Logic Update Final PLC Program
   "AON_PROCESS_BOOL" AT %M1000.3 : Bool;   // Logic Discuss With Process
   "AON_SCS_BOOL" AT %M1000.2 : Bool;   // Logic From SCS Update
   "AON_SITE_BOOL" AT %M1000.1 : Bool;   // Bypass to check at Commissioning
   "AOFF_SITE_BOOL" AT %M1000.0 : Bool;   // Bypass to check at Commissioning
   "OB35_CyclTime" AT %MW112 : Int;   // OB35 Cycle Time (100ms For PIDs)
   "_997CD100G02_FBY92" AT %M1055.5 : Bool;   // Select Carbon Safety Feed Pump
   "_997CD100G02_FBY91" AT %M1055.4 : Bool;   // Select Carbon Transfer Pump Path
   "_997CD100G02_FBGON" AT %M1055.3 : Bool;   // Group ON
   "_997CD100G01_FBY91" AT %M1055.2 : Bool;   // Select Fan E/W Exhaust / Dust Collector
   "_997CD100G04_FBI93" AT %MD3218 : Real;   // Time SP Strip Pro Scale Out Min
   "_997CD100G04_FBI92" AT %MD3214 : Real;   // Time SP Strip Pro 3 To 6 Hrs PV
   "_997CD100G04_FBI91" AT %MD3210 : Real;   // Counter Memory
   "_997CD100G04_FBGON" AT %M1057.2 : Bool;   // Group On
   "_997CD100G04_FBGOFF" AT %M1057.1 : Bool;   // Group Off
   "_997CD100G03B06_FBY91" AT %M1057.0 : Bool;   // Force Off
   "_997CD100G03B04_FBY91" AT %M1056.7 : Bool;   // Force Off
   "_997CD100G03B03_FBY91" AT %M1056.6 : Bool;   // Force Off
   "_997CD100G03B02_FBY91" AT %M1056.5 : Bool;   // Force Off
   "_997CD100G03B01_FBY91" AT %M1056.4 : Bool;   // Force Off
   "_997CD100G03B01_FBO1" AT %M1056.3 : Bool;   // Carbon Transfer From TK630 to TK640 seq Enabled
   "_997CD100G03_FBY93" AT %M1056.2 : Bool;   // Group Active
   "_997CD100G03_FBY92" AT %M1056.1 : Bool;   // Carbon Stripping Group Active
   "_997CD100G03_FBY91" AT %M1056.0 : Bool;   // Select Carbon Transfer
   "_997CD100G03_FBGON" AT %M1055.7 : Bool;   // Group On
   "_997CD100G03_FBGOFF" AT %M1055.6 : Bool;   // Group Off
   "_997CD100G04B01_FBY91" AT %M1058.6 : Bool;   // CT TK630 To TK640 Seq Enabled
   "_997CD100G04_FBY99" AT %M1058.5 : Bool;   // CNT02 Count Up
   "_997CD100G04_FBY98" AT %M1058.4 : Bool;   // CNT01 Count Up
   "_997CD100G04_FBY97" AT %M1058.3 : Bool;   // CNT02 Value Reach Zero
   "_997CD100G04_FBY96" AT %M1058.2 : Bool;   // CNT01 Value Reach Zero
   "_997CD100G04_FBY95" AT %M1058.1 : Bool;   // Sequence Group On
   "_997CD100G04_FBY94" AT %M1058.0 : Bool;   // Strip Pro 3 To 6 Hrs Delay
   "_997CD100G04_FBY93" AT %M1057.7 : Bool;
   "_997CD100G04_FBY92" AT %M1057.6 : Bool;   // Group Active
   "_997CD100G04_FBY91" AT %M1057.5 : Bool;   // Select Acid Wash / Pump Strip
   "_997CD100G04_FBY90" AT %M1057.4 : Bool;   // Select Pump Strip
   "_997CD100G04_FBY100" AT %M1057.3 : Bool;   // Strip Pro Timer Start IN
   "_997CD100G04_FBI97" AT %MW3234 : Int;   // CNT01 PV
   "_997CD100G04_FBI96" AT %MD3230 : Real;   // CNT01 Memory
   "_997CD100G04_FBI95" AT %MD3226 : Real;   // CNT01 Setpoint
   "_997CD100G04_FBI94" AT %MD3222 : Real;   // Strip Remaining Time
   "_997CD100G04I11_FBY93" AT %M1060.6 : Bool;   // Trans_03
   "_997CD100G04I11_FBY92" AT %M1060.5 : Bool;   // Trans_02
   "_997CD100G04I11_FBY91" AT %M1060.4 : Bool;   // Trans_01
   "_997CD100G04I11_FBY108" AT %M1060.3 : Bool;   // Unit Fault TK630 and TK640
   "_997CD100G04I11_FBY107" AT %M1060.2 : Bool;   // Goto Step
   "_997CD100G04I11_FBY106" AT %M1060.1 : Bool;   // Trans_16
   "_997CD100G04I11_FBY105" AT %M1060.0 : Bool;   // Trans_15
   "_997CD100G04I11_FBY104" AT %M1059.7 : Bool;   // Trans_14
   "_997CD100G04I11_FBY103" AT %M1059.6 : Bool;   // Trans_13
   "_997CD100G04I11_FBY102" AT %M1059.5 : Bool;   // Trans_12
   "_997CD100G04I11_FBY101" AT %M1059.4 : Bool;   // Trans_11
   "_997CD100G04I11_FBY100" AT %M1059.3 : Bool;   // Trans_10
   "_997CD100G04B04_FBY91" AT %M1059.2 : Bool;   // Valve Open / Close
   "_997CD100G04B03_FBY91" AT %M1059.1 : Bool;   // Valve Open / Close
   "_997CD100G04B02_FBY91" AT %M1059.0 : Bool;   // Valve Open / Close
   "_997CD100G04B01_FBY92" AT %M1058.7 : Bool;   // Force Off
   "_997CD100G05_FBI92" AT %MD3256 : Real;   // Y09 Time Delay
   "_997CD100G05_FBI91" AT %MD3252 : Real;   // Y02 Time Delay
   "_997CD100G04I12_FBY92" AT %M1061.7 : Bool;   // Trans_02
   "_997CD100G04I12_FBY91" AT %M1061.6 : Bool;   // Trans_01
   "_997CD100G04I12_FBRST" AT %M1061.5 : Bool;   // Sequence Reset
   "_997CD100G04I12_FBI94" AT %MD3248 : Real;   // Water Target level
   "_997CD100G04I12_FBI93" AT %MD3244 : Real;   // Saved Level Before Process Start
   "_997CD100G04I12_FBI92" AT %MD3240 : Real;   // NaOH Target Level
   "_997CD100G04I12_FBI91" AT %MD3236 : Real;   // NaOH Target Level Temp
   "_997CD100G04I11_FBY99" AT %M1061.4 : Bool;   // Trans_09
   "_997CD100G04I11_FBY98" AT %M1061.3 : Bool;   // Trans_08
   "_997CD100G04I11_FBY97" AT %M1061.2 : Bool;   // Trans_07
   "_997CD100G04I11_FBY96" AT %M1061.1 : Bool;   // Trans_06
   "_997CD100G04I11_FBY95" AT %M1061.0 : Bool;   // Trans_05
   "_997CD100G04I11_FBY94" AT %M1060.7 : Bool;   // Trans_04
   "1" AT %M0.1 : Bool;   // Constant High
   "0" AT %M0.0 : Bool;   // Constant Low
   "_2010CV300U01S11" AT %MD3034 : Real;   // Speed Setpoint
   "_2010CV300U01S01" AT %MD3030 : Real;   // Speed
   "_2010CV300U01J01" AT %MD3026 : Real;   // Power
   "_2010CV300U01I01" AT %MD3022 : Real;   // Current
   "Force 0" AT %M0.6 : Bool;   // Always FALSE, commissioning flag
   "Force 1" AT %M0.7 : Bool;   // Always TRUE, commissioning flag
   "_2010CV300U01C53" AT %M1003.0 : Bool;   // Local Stop
   "_2010CV300U01C51" AT %M1003.1 : Bool;   // Local Start
   "_2010CV300U01C73" AT %M1003.2 : Bool;   // Unbalance
   "_2010CV300U01C42" AT %M1003.3 : Bool;   // Drive / MCC Ready
   "_2010CV300U01C71" AT %M1003.4 : Bool;   // Motor Stalled
   "_2010CV300U01C45" AT %M1003.5 : Bool;   // Drawer Test Pos.
   "_2010CV300U01U41" AT %M1003.6 : Bool;   // General Fault
   "_2010CV300U01C44" AT %M1003.7 : Bool;   // Overload
   "_2010CV300U01C46" AT %M1004.0 : Bool;   // Bus Fault
   "_2010CV300U01C47" AT %M1004.1 : Bool;   // Drawer Oper. Pos.
   "_2010CV300U01C72" AT %M1004.2 : Bool;   // Earth Fault
   "_2010CV300U01C74" AT %M1004.3 : Bool;   // Reset Ack.
   "_2010CV300U01U42" AT %M1004.4 : Bool;   // General Warning
   "_2010CV300U01C56" AT %M1004.5 : Bool;   // Safety Switch
   "_2010CV300U01C61" AT %M1004.6 : Bool;   // Return
   "M_BC180_GS" AT %M1000.6 : Bool;
   "M_BC120_GS" AT %M1000.7 : Bool;
   "_2010LV100P01C61" AT %I6159.0 : Bool;
END_VAR

VAR_GLOBAL   // PLC tag table "asutp"
   "sim_on" AT %M2000.0 : Bool;
   "_997CD100G03_alarm_warning" AT %M1016.4 : Bool;   // m1016.4
   "_2010SJ950M01_O1" AT %M1100.0 : Bool;
   "_2010SJ950M01_O1_Q" AT %M1100.1 : Bool;
   "_2010SJ950M01_O2" AT %M1100.2 : Bool;
   "_2010SJ950M01_O2_Q" AT %M1100.3 : Bool;
   "_2010SJ950M01_F1_Q1" AT %M1100.4 : Bool;
   "_2010SJ950M01I01" AT %MD4580 : Real;
   "_2010SJ950M01C44" AT %M1100.5 : Bool;
   "_2010SJ950M01C61" AT %M1100.6 : Bool;
   "_2010SJ950M01C51" AT %M1100.7 : Bool;
   "_2010SJ950M01C53" AT %M1101.0 : Bool;
   "_2010SJ950M01C74" AT %M1101.1 : Bool;
   "_2010SJ950M01C42" AT %M1101.2 : Bool;
   "_2010SJ950M01C71" AT %M1101.3 : Bool;
   "_2010SJ950M01C72" AT %M1101.4 : Bool;
   "_2010SJ950M01C73" AT %M1101.5 : Bool;
   "_2010SJ950M01U41" AT %M1101.6 : Bool;
   "_2010SJ950M01U42" AT %M1101.7 : Bool;
   "_2010SJ950M01C46" AT %M1102.0 : Bool;
   "_2010SJ950M01C47" AT %M1102.1 : Bool;
   "_2010SJ950M01C45" AT %M1102.2 : Bool;
   "tag77" AT %M9000.2 : Bool;
   "tag79" AT %M9000.3 : Bool;
   "tag80" AT %MD9004 : Real;
END_VAR

VAR_GLOBAL   // PLC tag table "PCM"
   "PMC_YSH_400V" AT %I0.0 : Bool;   // PMC Healthy 400V (1=ok)
   "PMC_YSQ_10QG01" AT %I0.1 : Bool;   // PMC Breaker Feedback Main PMC (1=ok)
   "PMC_YSQ_10Q03" AT %I0.2 : Bool;   // PMC Breaker Feedback Control (1=ok)
   "SPARE_PMC_1_DI1_3" AT %I0.3 : Bool;   // PMC spare
   "PMC_YSQ_20Q03" AT %I0.4 : Bool;   // PMC Breaker Feedback 230V Electronic (1=ok)
   "PMC_YSQ_20Q04" AT %I0.5 : Bool;   // PMC Breaker Feedback 230V Control (1=ok)
   "PMC_YSQ_26Q01" AT %I0.6 : Bool;   // PMC Breaker Feedback 24V Safety relay (1=ok)
   "PMC_YSQ_30Q02" AT %I0.7 : Bool;   // PMC Breaker Feedback 230V Utility (1=ok)
   "PMC_YSQ_30Q03" AT %I1.0 : Bool;   // PMC Breaker Feedback 230V Safety relay (1=ok)
   "PMC_US_UPS" AT %I1.1 : Bool;   // PMC Power on return UPS (1=ok)
   "PMC_OA3" AT %I1.2 : Bool;   // PMC Emergency stop PB Box (1=ok)
   "PMC_YSES_50FES01" AT %I1.3 : Bool;   // PMC Safety relay feedback (1=ok)
   "PMC_OA" AT %I1.4 : Bool;   // PMC Emergency stop PB (1=ok)
   "Feed110_YSQ" AT %I1.5 : Bool;   // Feeder BF110 Breaker Feedback (1=ok)
   "Feed110_OA" AT %I1.6 : Bool;   // Feeder BF110 Pull Rope (1=ok)
   "Feed110_HGL3" AT %I1.7 : Bool;   // Feeder BF110 Local/Remote selector Box (1=remote)
   "Feed110_HSST3" AT %I2.0 : Bool;   // Feeder BF110 Push button start Box (1 pulse)
   "Feed110_HSSP3" AT %I2.1 : Bool;   // Feeder BF110 Push button stop Box (0 pulse)
   "Feed110_OA3" AT %I2.2 : Bool;   // Feeder BF110 Emergency stop PB Box (1=ok)
   "Feed110_HGR3" AT %I2.3 : Bool;   // Feeder BF110 Forcing red traffic light Box (1=red)
   "Feed110_HSH3" AT %I2.4 : Bool;   // Feeder BF110 Speed setpoint increase Box (1 pulse)
   "Feed110_HSL3" AT %I2.5 : Bool;   // Feeder BF110 Speed setpoint decrease Box (1 pulse)
   "Conv120_YSQ" AT %I2.6 : Bool;   // Conveyor CV120 Breaker Feedback (1=ok)
   "Conv120_YSK" AT %I2.7 : Bool;   // Conveyor CV120 Contactor feedback (1=closed)
   "Conv120_OA" AT %I3.0 : Bool;   // Conveyor CV120 Emergency stop PB (1=ok)
   "Conv120_GS" AT %I3.1 : Bool;   // Conveyor CV120 Rotation control sensor (1 pulse)
   "Scrn130_YSQ" AT %I3.2 : Bool;   // Screen SC130 Breaker Feedback (1=ok)
   "Scrn130_TSH_BREAK" AT %I3.3 : Bool;   // Screen SC130 High temperature breake (1=ok)
   "Scrn130_OA" AT %I3.4 : Bool;   // Screen SC130 Emergency stop PB (1=ok)
   "Crus150_YSQ" AT %I3.5 : Bool;   // Crusher CR150 Breaker Feedback (1=ok)
   "Crus150_YSK" AT %I3.6 : Bool;   // Crusher CR150 Contactor feedback (1=closed)
   "Crus150_YAA" AT %I3.7 : Bool;   // Crusher CR150 SS fault (1=ok)
   "Crus150_YSS" AT %I4.0 : Bool;   // Crusher CR150 SS end of start (1=closed)
   "Crus150_NS" AT %I4.1 : Bool;   // Crusher CR150 PTC sensor (1=ok)
   "Pump150A1_YSQ" AT %I4.2 : Bool;   // Pump CR150 Breaker Feedback (1=ok)
   "Crus150_OA" AT %I4.3 : Bool;   // Crusher CR150 Emergency stop PB (1=ok)
   "Pump150A1_YS_Q1" AT %I4.4 : Bool;   // Pump CR150 Feedback main Switch Q1 (1=closed)
   "Pump150A1_YSK_Q9" AT %I4.5 : Bool;   // Pump CR150 Contactor feedback hydrau pump Q9 (1=started)
   "Pump150A1_PSL_B92" AT %I4.6 : Bool;   // Pump CR150 Low pressure switch clamping press B92/K92 (1=ok)
   "Pump150A1_YS_K96" AT %I4.7 : Bool;   // Pump CR150 Feedback setting lightening K96 (1=started)
   "Feed110_OA1" AT %I5.0 : Bool;   // ???
   "Pump150A1_LSL_B93" AT %I5.1 : Bool;   // Pump CR150 Low level switch oil B93/KL (1=alm)
   "Pump150A1_XS_B95" AT %I5.2 : Bool;   // Pump CR150 Clogging filter sensor B95/KF (1=alm)
   "Pump150A1_PSL_B91" AT %I5.3 : Bool;   // Pump CR150 Low pressure switch oil B91/KP (1=alm)
   "Conv180_YSQ" AT %I5.4 : Bool;   // Conveyor CV180 Breaker Feedback (1=ok)
   "Conv180_YSK" AT %I5.5 : Bool;   // Conveyor CV180 Contactor feedback (1=closed)
   "Conv180_YAA" AT %I5.6 : Bool;   // Conveyor CV180 SS fault (1=ok)
   "Conv180_YSS" AT %I5.7 : Bool;   // Conveyor CV180 SS end of start (1=closed)
   "Conv180_YAT" AT %I6.0 : Bool;   // Conveyor CV180 Thermal breaker fault (0=ok)
   "Conv180_OAC" AT %I6.1 : Bool;   // Conveyor CV180 Emergency stop cord (1=ok)
   "Conv180_LSHH" AT %I6.2 : Bool;   // Conveyor CV180 Blocked chute (1=ok)
   "Conv180_GS" AT %I6.3 : Bool;   // Conveyor CV180 Rotation control sensor (1 pulse)
   "Conv300_WS" AT %I6.4 : Bool;   // Conveyor CV300 Beltscale flow switch Production pulse (1 pulse)
   "Conv300_WT_RDY" AT %I6.5 : Bool;   // Conveyor CV300 Beltscale ready
   "Conv180_YS_TARE2" AT %I6.6 : Bool;   // Conveyor CV180 Feedback Tare 2 (1=closed)
   "Ovbd190_YSQ" AT %I6.7 : Bool;   // Overband OV190 Breaker Feedback PMC (1=ok)
   "Ovbd190_YSK" AT %I7.0 : Bool;   // Overband OV190 Contactor feedback PMC (1=closed)
   "Ovbd190_YSK3" AT %I7.1 : Bool;   // Overband OV190 Contactor feedback Box (1=closed)
   "Ovbd190_YSH3" AT %I7.2 : Bool;   // Overband OV190 Healthy Box (1=ok)
   "SPARE_PMC_1_DI4_11" AT %I7.3 : Bool;   // PMC spare
   "Ovbd190_SW3" AT %I7.4 : Bool;   // Overband OV190 Isolator switch Box (1=closed)
   "Ovbd190_OA3" AT %I7.5 : Bool;   // Overband OV190 Emergency stop PB Box (1=ok)
   "Ovbd190_YSES" AT %I7.6 : Bool;   // Overband OV190 Safety relay feedback (1=ok)
   "Conv300_YP" AT %I7.7 : Bool;   // Conveyor CV300 Start permissive running autorisation (1=ok)
   "Conv300_OA" AT %I8.0 : Bool;   // Conveyor CV300 Emergency stop PB (1=ok)
   "Feed110_YSQ_Heater" AT %I8.1 : Bool;   // PMC spare
   "SPARE_PMC_1_DI5_2" AT %I8.2 : Bool;   // PMC spare
   "SPARE_PMC_1_DI5_3" AT %I8.3 : Bool;   // PMC spare
   "SPARE_PMC_1_DI5_4" AT %I8.4 : Bool;   // PMC spare
   "PMC_YSQ_42Q02" AT %I8.5 : Bool;   // PMC spare
   "SPARE_PMC_1_DI5_6" AT %I8.6 : Bool;   // PMC spare
   "SPARE_PMC_1_DI5_7" AT %I8.7 : Bool;   // PMC spare
   "SPARE_PMC_1_DI5_8" AT %I9.0 : Bool;   // PMC spare
   "SPARE_PMC_1_DI5_9" AT %I9.1 : Bool;   // PMC spare
   "SPARE_PMC_1_DI5_10" AT %I9.2 : Bool;   // PMC spare
   "SPARE_PMC_1_DI5_11" AT %I9.3 : Bool;   // PMC spare
   "SPARE_PMC_1_DI5_12" AT %I9.4 : Bool;   // PMC spare
   "SPARE_PMC_1_DI5_13" AT %I9.5 : Bool;   // PMC spare
   "SPARE_PMC_1_DI5_14" AT %I9.6 : Bool;   // PMC spare
   "SPARE_PMC_1_DI5_15" AT %I9.7 : Bool;   // PMC spare
   "PMC_YUZES_50FES01" AT %Q0.0 : Bool;   // PMC Safety relay reset (1 pulse)
   "Conv120_ALH" AT %Q0.1 : Bool;   // Conveyor CV120 Horn
   "Conv120_ALF" AT %Q0.2 : Bool;   // Conveyor CV120 Flashing light
   "Hopp100_OLG" AT %Q0.3 : Bool;   // Hopper HP100 Green traffic light
   "Hopp100_OLR" AT %Q1.0 : Bool;   // Hopper HP100 Red traffic light
   "Feed110_OLL3" AT %Q1.1 : Bool;   // Feeder BF110 Local mode light Box
   "Conv120_YCK" AT %Q1.2 : Bool;   // Conveyor CV120 Contactor start order
   "Crus150_YCA" AT %Q1.3 : Bool;   // Crusher CR150 SS start order (1=start)
   "Pump150A1_YS" AT %Q2.0 : Bool;   // Pump CR150 Feedback crusher started (1=started)
   "Conv180_YCA" AT %Q2.1 : Bool;   // Conveyor CV180 SS start order (1=start)
   "Conv180_YC_Tare" AT %Q2.2 : Bool;   // Conveyor CV180 Start order Tare
   "Ovbd190_YC3" AT %Q2.3 : Bool;   // Overband OV190 Start order Box
   "PMC_Reset_Q42Q02" AT %Q3.0 : Bool;   // PMC spare
   "SPARE_PMC_1_DO4_1" AT %Q3.1 : Bool;   // PMC spare
   "SPARE_PMC_1_DO4_2" AT %Q3.2 : Bool;   // PMC spare
   "SPARE_PMC_1_DO4_3" AT %Q3.3 : Bool;   // PMC spare
   "Hopp100_LT" AT %IW256 : Int;   // Hopper HP100 Level transmitter primary hopper (0-100%)
   "Feed110_GT" AT %IW258 : Int;   // Feeder BF110 GT (0-100%)
   "Crus150_IT" AT %IW260 : Int;   // Crusher CR150 Current transmitter (0-[TI setting]A)
   "Crus150_LT" AT %IW262 : Int;   // Crusher CR150 Level transmitter (0-100%)
   "Conv300_WT_flow" AT %IW264 : Int;   // Conveyor CV300 Beltscale flow transmitter (0-[MAX]tph)
   "Conv300_WT_speed" AT %IW266 : Int;   // Conveyor CV300 Beltscale speed transmitter (0-[MAX]ms)
   "SPARE_AI270" AT %IW270 : Int;   // Spare
   "_2010CV300D06Z41" AT %I10.4 : Bool;   // Sway Max 1 Left
   "SPARE_DI11_1" AT %I11.1 : Bool;   // Spare
   "SPARE_DI11_2" AT %I11.2 : Bool;   // Spare
   "_2010SJ950D01L41" AT %I10.0 : Bool;   // Level Max
   "_2010WG016N01U41" AT %I10.1 : Bool;   // General Fault
   "_2010WG016N01Q41" AT %I10.2 : Bool;   // Quantity Pulse
   "_2010CV300D01S41" AT %I10.3 : Bool;   // Speed Min
   "_2010CV300D06Z42" AT %I10.5 : Bool;   // Sway Max 1 Right
   "_2010CV300D06Z44" AT %I10.6 : Bool;   // Sway Max 2 Left
   "_2010CV300D06Z45" AT %I10.7 : Bool;   // Sway Max 2 Right
   "_2010CV300D06Z43" AT %I11.0 : Bool;   // Belt Rip Detection
   "_2010CV300D12Z41" AT %I11.3 : Bool;   // Продольный порез ленты
   "_2010CV300D13Z41" AT %I11.4 : Bool;   // Pos. Open
   "_2010CV300D14Z41" AT %I11.5 : Bool;   // Pos. Open
   "_2010CV300D15Z41" AT %I11.6 : Bool;   // Pos. Open
   "_2010CV300D17Z41" AT %I11.7 : Bool;   // Pos. Open
END_VAR

VAR_GLOBAL   // PLC tag table "CV300VFD"
   "CV300_VFD_ SB_Running_State" AT %IB509 : Byte;
   "SW Bus Volt Estab" AT %I508.0 : Bool;   // 1 - Rdy To Run
   "SW Mtr Grp feedback M1" AT %I508.1 : Bool;
   "SW Mtr Grp feedback M2" AT %I508.2 : Bool;
   "SW Mtr Type Feedback" AT %I508.3 : Bool;   // 1 - Synchronus; 2 - Asynchronus.
   "SW Overload Pre Alrm feedback" AT %I508.4 : Bool;
   "SW Run Stop Mode1" AT %I508.5 : Bool;   // 0:0 - Keypad Crl; 1:0 - Termenal Crl
   "SW Run Stop Mode2" AT %I508.6 : Bool;   // 0:1 - Comm Crl
   "SW HeartBeat" AT %I508.7 : Bool;
   "Actual Speed" AT %IW510 : Int;   // *100Hz
   "Motor Power" AT %IW512 : Int;   // *10 %
   "Motor Current" AT %IW516 : Int;   // * 20 A
   "Last Fault Word" AT %IW520 : Word;
   "Last Warning Word" AT %IW522 : Word;
   "CW Cmd" AT %QB509 : Byte;   // 1- FRun; 2 - RRun; 3 - FJg; 4 - RJg; 5 - Stp; 6 - EmStp; 7 - Flt Rst; 8 - Stp Jg;
   "CW EnWrt" AT %Q508.0 : Bool;
END_VAR

VAR_GLOBAL   // PLC tag table "997CS110A01"
   "_2015PU027Y01Z41" AT %I1022.0 : Bool;   // Aspiration Level Control Valve, Pos. Open
   "_2015PU027Y01Z42" AT %I1022.1 : Bool;   // Aspiration Level Control Valve, Pos. Closed
   "_2015PU028Y01Z41" AT %I1022.2 : Bool;   // Aspiration Bypass Water Valve, Pos. Open
   "_2015PU028Y01Z42" AT %I1022.3 : Bool;   // Aspiration Bypass Water Valve, Pos. Closed
   "_2010UP100G01U41" AT %I1024.4 : Bool;   // UPC Low Battery
   "_2010UP100G01U42" AT %I1024.5 : Bool;   // UPC Summary Alarm
   "_2015SU026N01L01" AT %IW1006 : Word;
   "_2015SU026N02F01" AT %IW1008 : Word;
   "_2015PU027N01L01" AT %IW1010 : Word;
   "_2015PU027Y01C31" AT %Q1008.0 : Bool;   // Aspiration Level Control Valve, Command
   "_2015PU028Y01C31" AT %Q1008.1 : Bool;
END_VAR

TYPE "ACESYS_ADPT_PFISTERSDD"
TITLE = Data Structure for Adaptor block (data exchange with HMI)
AUTHOR : FLSmidth
FAMILY : ACESYS
NAME : ADPT
VERSION : 8.0
   STRUCT
      Intell_Type : Int;
      VersionNo : Int;
      BuildNo : Int;
      FuncType : Int;
      Options : Int;
      NetNo : Int;
      NodeNo : Int;
      Sim_Enable : Bool;   // Device Simulation Enabled
      SpareBool07 : Bool;
      SpareBool06 : Bool;
      SpareBool05 : Bool;
      SpareBool04 : Bool;
      SpareBool03 : Bool;
      SpareBool02 : Bool;
      SpareBool01 : Bool;
      MessageID : Byte;
      DosingMode : Bool;
      MeasuringMode : Bool;
      FieldMode : Bool;
      Run : Bool;
      CorrectionDone : Bool;
      ToltalizerPulse : Bool;
      SelectVals : Bool;
      Togglebit_R : Bool;
      Feedrate : Int;
      Speed : Int;
      Load : Int;
      Preload : Int;
      Current : Int;
      Droppointload : Int;
      SpareByte : Byte;
      CmdDosingMode : Bool;
      CmdMeasuringMode : Bool;
      CmdStart : Bool;
      CmdAcknowledge : Bool;
      CmdCorrection : Bool;
      SpareBool : Bool;
      CmdSelectVals : Bool;
      Togglebit_T : Bool;
      DosingSetpoint : Int;
      SpeedSetpoint : Int;
      RemoteCorrection : Int;
   END_STRUCT;
END_TYPE

TYPE "ACESYS_PLCToPLC_H"
TITLE = PLC to PLC Communication Data Layout
AUTHOR : FLSmidth
FAMILY : ACESYS
NAME : PLCtoPLC
VERSION : 8.0
   STRUCT
      Watchdog : Bool;   // Watchdog Bit
      Simulation_Enabled : Bool;   // Device Simulation Enabled
      Spare_2 : Bool;   // Not Used
      Spare_3 : Bool;   // Not Used
      Spare_4 : Bool;   // Not Used
      Spare_5 : Bool;   // Not Used
      Spare_6 : Bool;   // Not Used
      Spare_7 : Bool;   // Not Used
      BOOLEAN : Array[0..63] of Bool;   // Boolean Data
      REAL_VAL : Array[0..15] of Real;   // Real Data
      INT_VAL : Array[0..15] of Int;   // Interger Data
      H_PLC_STATUS : Struct
         CPU00_MASTER : Bool;
         CPU01_MASTER : Bool;
         CPU00_RUN : Bool;
         CPU01_RUN : Bool;
         Redundancy_State : Bool;
         Conn1_RECV_Error : Bool;
         Conn2_RECV_Error : Bool;
         Conn3_RECV_Error : Bool;
         Conn4_RECV_Error : Bool;
         Sapre_1 : Bool;
         Sapre_2 : Bool;
         Sapre_3 : Bool;
         Sapre_4 : Bool;
         Sapre_5 : Bool;
         Sapre_6 : Bool;
         CURR_Connection : Int;
      END_STRUCT;
   END_STRUCT;
END_TYPE

TYPE "ACESYS_ADPT_SCHENCK"
   STRUCT
      Info : Struct
         Intell_Type : Int;
         VersionNo : Int;
         BuildNo : Int;
         FuncType : Int;
         Options : Int;
         NetNo : Int;
         NodeNo : Int;
         Sim_Enable : Bool;   // Device Simulation Enabled
         BusFault : Bool;
         FuncTypeErr : Bool;
         ScaleTypeErr : Bool;
         SpareBool5 : Bool;
         SpareBool6 : Bool;
         SpareBool7 : Bool;
         SpareBool8 : Bool;
         SpareBool9 : Bool;
         SpareBool10 : Bool;
         SpareBool11 : Bool;
         SpareBool12 : Bool;
         SpareBool13 : Bool;
         SpareBool14 : Bool;
         SpareBool15 : Bool;
         SpareBool16 : Bool;
         SpareInt1 : Int;
         SpareInt2 : Int;
         SpareInt3 : Int;
         SpareInt4 : Int;
         SpareInt5 : Int;
         SpareIntReal1 : Real;
         SpareIntReal2 : Real;
         SpareIntReal3 : Real;
         SpareIntReal4 : Real;
         SpareIntReal5 : Real;
      END_STRUCT;
      Rx : Struct
         SB00_0_NormMode : Bool;   // Normal Mode
         SB00_1_KBMode : Bool;   // Keyboard Mode
         SB00_2_LocMode : Bool;   // Local Mode
         SB00_3_SimMode : Bool;   // Simulation Mode
         SB00_4 : Bool;   // Volum. Start-Up
         SB00_5 : Bool;   // Meas. Drive On
         SB00_6 : Bool;   // Wheel Meas. Drive Delay
         SB00_7 : Bool;   // Setpoint Limited
         SB01_0_ScaleOn : Bool;   // Scale On (RET)
         SB01_1_NotRel : Bool;   // Not Released
         SB01_2 : Bool;   // Counter Active
         SB01_3_VolMode : Bool;   // Volumetric Mode
         SB01_4 : Bool;   // Select Langugage Ok
         SB01_5_Alarm : Bool;   // Alarm
         SB01_6_Warn : Bool;   // Warning
         SB01_7_CalActive : Bool;   // Calibration Active
         SB02_0 : Bool;   // Tare
         SB02_1 : Bool;   // Zero Set
         SB02_2 : Bool;   // Weight Check
         SB02_3 : Bool;   // Pulses/Revolution
         SB02_4 : Bool;   // DAE Adjustment
         SB02_5 : Bool;   // Auto Zero Active
         SB02_6 : Bool;   // Volumetric Adaption
         SB02_7 : Bool;   // Gravimetric Optimization
         SB03_0 : Bool;   // Batch Selected
         SB03_1 : Bool;   // Batch Active
         SB03_2 : Bool;   // Batch Dribble Feed (Pre-act Cont.)
         SB03_3 : Bool;   // Batch + Clearance
         SB03_4 : Bool;   // NON-SI Active
         SB03_5 : Bool;   // Dead Time Active
         SB03_6 : Bool;   // Dead Time Setpoint Active
         SB03_7 : Bool;   // Dead Time ON/OFF Active
         SD04_FeedRate : Real;   // Feed Rate [kg/h]
         SD08_Totalizer1 : Real;   // Totalizer 1 [kg]
         SD12_BinWeight : Real;   // Bin Weigher Fill Weight [kg]
         SB16_SoftRev : Byte;   // Software Revision
         SB17_ScaleType : Byte;   // Scale Type
         SW18_SoftVer : Word;   // Software Version
         SB20_0 : Bool;   // KME Active
         SB20_1 : Bool;   // No Alarm
         SB20_2 : Bool;   // No Warning
         SB20_3 : Bool;   // Pulse counter reading
         SB20_4_NoDev : Bool;   // No Deviation
         SB20_5_Ready : Bool;   // Ready
         SB20_6 : Bool;   // KME Rel Tare Not Exceeded
         SB20_7 : Bool;   // KME Abs. Tare Not Exceeded
         SB21_0 : Bool;   // Calibr. Set Norminal Feed Rate
         SB21_1 : Bool;   // Pre-cut-off amount Dig. Output
         SB21_2 : Bool;   // MAX Limit Value
         SB21_3 : Bool;   // MIN Limit Value
         SB21_4 : Bool;   // VSM 20110 (DISOCONT L)
         SB21_5 : Bool;   // Make-up active
         SB21_6 : Bool;   // VSM 20107 (pulverized coal)
         SB21_7_FillBin : Bool;   // Fill Bin Weigher
         SB22 : Byte;   // Standby
         SB23_0 : Bool;   // KME Rel. Range Not Exceeded
         SB23_1 : Bool;   // KME Abs. Range Not Exceeded
         SB23_2 : Bool;   // VSM Type A (big)
         SB23_3 : Bool;   // VSM Type F (fast)
         SB23_4 : Bool;
         SB23_5 : Bool;
         SB23_6 : Bool;
         SB23_7 : Bool;
         SB24_EventHI : Byte;   // Highest-Priority Event (HI)
         SB25_EventLO : Byte;   // Highest-Priority Event (LO)
         SB26 : Byte;   // Number in parameter block
         SB27 : Byte;   // Parameter block including the event class
         SD28 : Real;   // User selected parameter from faceplate
         SB32_0 : Bool;   // Feed Rate > Max
         SB32_1 : Bool;   // Feed Rate < Min
         SB32_2 : Bool;   // Belt Load > Max
         SB32_3 : Bool;   // Belt Load < Min
         SB32_4 : Bool;   // Speed > Max
         SB32_5 : Bool;   // Speed < Min
         SB32_6 : Bool;   // Bin > Max
         SB32_7 : Bool;   // Bin < Min
         SB33_0 : Bool;   // Meas. System
         SB33_1 : Bool;   // Gain-In-Weight
         SB33_2 : Bool;   // Filling Active
         SB33_3_Discharge : Bool;   // Discharge Active
         SB33_4 : Bool;   // Gate Open
         SB33_5 : Bool;   // Gate Closed
         SB33_6 : Bool;   // 2nd Batch Unit Active (VLW20151 only)
         SB33_7_Hopper : Bool;   // Surge Hopper present
         SB34_0_CheckAvail : Bool;   // 8 - Check System Available
         SB34_1_RelTaraExc : Bool;   // Rel. tare Exceeded
         SB34_2_AbsTaraExc : Bool;   // Abs. tare Exceeded
         SB34_3_RelRangeExc : Bool;   // Rel. range Exceeded
         SB34_4_AbsRangeExc : Bool;   // Abs. range Exceeded
         SB34_5 : Bool;   // Check Meas. Announced
         SB34_6_Prepare : Bool;   // Prepare Check
         SB34_7_CheckActive : Bool;   // Check Active
         SB35_0 : Bool;   // Bin Level Control existent
         SB35_1 : Bool;   // Hopper level > Max
         SB35_2 : Bool;   // Hopper level < Min
         SB35_3 : Bool;   // Measured load > Max
         SB35_4 : Bool;   // Measured load < Min
         SB35_5 : Bool;   // n > Max
         SB35_6 : Bool;   // n < Min
         SB35_7_CheckWaitAck : Bool;   // Check System waits for acknowledgement
         SD36_CheckResult : Real;   // Check Result F/Z [Factor] 1=0%
         SD40_ActSP : Real;   // Actual Setpoint [kg/h]
         SD44_Deviation : Real;   // Deviation
         SD48 : Real;   // Not Used
         SD52 : Real;   // Not Used
      END_STRUCT;
      Tx_C : Struct
         CW00 : Int;   // Command ID 1: Command 4+5 (140 Hex / 320 Dec)
         CB02_0 : Bool;   // Command 4 (HI): Volm. Synchronous
         CB02_1 : Bool;   // Command 4 (HI): Moisture Corr. On
         CB02_2 : Bool;   // Command 4 (HI): Moisture Corr. Off
         CB02_3 : Bool;   // Command 4 (HI): Meas. Drive Off
         CB02_4 : Bool;   // Command 4 (HI): Gate Feedback
         CB02_5 : Bool;   // Command 4 (HI): Open Gate Manual
         CB02_6 : Bool;   // Command 4 (HI): Stop Gate Manual
         CB02_7 : Bool;   // Command 4 (HI): Close Gate Manual
         CB03_0_StrScale : Bool;   // Command 4 (LO): Start Scale
         CB03_1_StpScale : Bool;   // Command 4 (LO): Stop Scale
         CB03_2_ClearEvent : Bool;   // Command 4 (LO): Clear Events (RESET)
         CB03_3_Release : Bool;   // Command 4 (LO): Release
         CB03_4_SelVol : Bool;   // Command 4 (LO): Select Volumetric Mode
         CB03_5_SelGrav : Bool;   // Command 4 (LO): Select Gravimetric Mode
         CB03_6_ResTot : Bool;   // Command 4 (LO): Reset Totalizer 1
         CB03_7 : Bool;   // Command 4 (LO): Reset Totalizer 2
         CB04_0 : Bool;   // Command 5 (HI): Filling Start
         CB04_1 : Bool;   // Command 5 (HI): Filling Stop
         CB04_2 : Bool;   // Command 5 (HI): Emptying Start
         CB04_3 : Bool;   // Command 5 (HI): Emptying Stop
         CB04_4 : Bool;   // Command 5 (HI): Init .Hopper Controller
         CB04_5 : Bool;   // Command 5 (HI): Activate Fill Unit
         CB04_6 : Bool;   // Command 5 (HI): Activate Prefeeder
         CB04_7 : Bool;   // Command 5 (HI): Stop Prefeeder
         CB05_0 : Bool;   // Command 5 (LO): Select Batch
         CB05_1 : Bool;   // Command 5 (LO): Deselect Batch
         CB05_2 : Bool;   // Command 5 (LO): Abort Batch
         CB05_3 : Bool;   // Command 5 (LO): Next Batch + Clearance
         CB05_4 : Bool;   // Command 5 (LO): Make-Up
         CB05_5 : Bool;   // Command 5 (LO): Emergency Setpoint On
         CB05_6 : Bool;   // Command 5 (LO): Emergency Setpoint Off
         CB05_7 : Bool;   // Command 5 (LO): Meas Drive On
         CW06 : Int;   // Command ID 2: Absolute Setpoint ID (250 Hex / 592 Dec)
         CD08_SP : Real;   // Absolute Setpoint [kg/h]
         CW12 : Int;   // Command ID 3: Command 6 + 7 (160 Hex / 352 Dec)
         CB14_0 : Bool;   // Command 6 (HI): Bin controller Autom.
         CB14_1 : Bool;   // Command 6 (HI): Bin controller Manual
         CB14_2 : Bool;   // Command 6 (HI): Bin controller Man. Start
         CB14_3 : Bool;   // Command 6 (HI): Bin controller Man Stop
         CB14_4 : Bool;   // Command 6 (HI): Optimization Bin Controller
         CB14_5 : Bool;   // Command 6 (HI): Print check Meas. Result
         CB14_6 : Bool;   // Command 6 (HI): Dead Time preassign
         CB14_7 : Bool;   // Command 6 (HI): Dead Time initialize
         CB15_0_StrTara : Bool;   // Command 6 (LO): Start internal check for tara
         CB15_1_StrRange : Bool;   // Command 6 (LO): Start internal check for range
         CB15_2_Acquire : Bool;   // Command 6 (LO): Acquire check result
         CB15_3_Cancel : Bool;   // Command 6 (LO): Cancel check measurement
         CB15_4 : Bool;   // Command 6 (LO): Release check system
         CB15_5 : Bool;   // Command 6 (LO): Acquire ext. corr. factor for tare
         CB15_6 : Bool;   // Command 6 (LO): Acquire ext. corr. factor for range
         CB15_7 : Bool;   // Command 6 (LO): Start external check
         CB16_0 : Bool;   // Command 7 (HI): Linearization P4
         CB16_1 : Bool;   // Command 7 (HI): Volmetric
         CB16_2 : Bool;   // Command 7 (HI): Optimize controller
         CB16_3 : Bool;   // Command 7 (HI): Calibration Acquire
         CB16_4 : Bool;   // Command 7 (HI): Calibration Abort
         CB16_5 : Bool;   // Command 7 (HI): Time Acquire
         CB16_6 : Bool;   // Command 7 (HI): Bin: Tare
         CB16_7 : Bool;   // Command 7 (HI): Bin: Weight Check
         CB17_0 : Bool;   // Command 7 (LO): Tare
         CB17_1 : Bool;   // Command 7 (LO): Zero Set
         CB17_2 : Bool;   // Command 7 (LO): Weight Check
         CB17_3 : Bool;   // Command 7 (LO): Pulses/Revolution
         CB17_4 : Bool;   // Command 7 (LO): DAE Adjustment
         CB17_5 : Bool;   // Command 7 (LO): Liniarization P1
         CB17_6 : Bool;   // Command 7 (LO): Liniarization P2
         CB17_7 : Bool;   // Command 7 (LO): Liniarization P3
      END_STRUCT;
      Tx_D : Struct
         CW18 : Int;   // Command ID 4: Command 10 + 11 (1A0 Hex / 416 Dec)
         CB20_0 : Bool;   // Command 10 (HI): Reset Sum of Component 9
         CB20_1 : Bool;   // Command 10 (HI): Reset Sum of Component 10
         CB20_2 : Bool;   // Command 10 (HI): Reset Sum of Batches
         CB20_3_FillStopped : Bool;   // Command 10 (HI): Filling Stopped
         CB20_4 : Bool;   // Command 10 (HI): Start (static)
         CB20_5 : Bool;   // Command 10 (HI):
         CB20_6 : Bool;   // Command 10 (HI): Activate 2nd Batch Unit
         CB20_7 : Bool;   // Command 10 (HI): De-activate 2nd Batch Unit
         CB21_0 : Bool;   // Command 10 (LO): Reset Sum of Component 1
         CB21_1 : Bool;   // Command 10 (LO): Reset Sum of Component 2
         CB21_2 : Bool;   // Command 10 (LO): Reset Sum of Component 3
         CB21_3 : Bool;   // Command 10 (LO): Reset Sum of Component 4
         CB21_4 : Bool;   // Command 10 (LO): Reset Sum of Component 5
         CB21_5 : Bool;   // Command 10 (LO): Reset Sum of Component 6
         CB21_6 : Bool;   // Command 10 (LO): Reset Sum of Component 7
         CB21_7 : Bool;   // Command 10 (LO): Reset Sum of Component 8
         CB22_0 : Bool;   // Command 11 (HI): Feeder 1 Active
         CB22_1 : Bool;   // Command 11 (HI): Feeder 1 Not Active
         CB22_2 : Bool;   // Command 11 (HI): Feeder 1 Active
         CB22_3 : Bool;   // Command 11 (HI): Feeder 1 Not Active
         CB22_4 : Bool;   // Command 11 (HI): Set Norminal Feed Rate
         CB22_5 : Bool;   // Command 11 (HI): Copy feed index block
         CB22_6 : Bool;   // Command 11 (HI):
         CB22_7 : Bool;   // Command 11 (HI):
         CB23 : Byte;   // Command 11 (LO): Component Number (1 Byte)
         CW24 : Int;   // Status ID 1: Totalizer 1 [kg] (752 Hex / 1874 Dec)
         CW26 : Int;   // Status ID 2: Bin Weigher Fill Weight [kg] (762 Hex / 1890 Dec)
         CW28 : Int;   // Status ID 3: Status 0 + 1 (2D0 Hex / 720 Dec)
         CW30 : Int;   // Status ID 4: Status 8 + 9 (350 Hex / 848 Dec)
         CW32 : Int;   // Status ID 5: Priority Event (610 Hex / 1552 Dec)
         CW34 : Int;   // Status ID 6: Varialbe ID from faceplate range 1872-2158 (dec)
         CW36 : Int;   // Status ID 7: Status 4 + 5 (310 Hex / 784 Dec)
         CW38 : Int;   // Status ID 8: Check Result F/Z (7EA Hex / 2026 Dec)
         CW40 : Int;   // Status ID 9: Actual Setpoint [kg/h] (766 Hex / 1894 Dec)
         CW42 : Int;   // Status ID 10: Deviation (770 Hex / 1904 Dec)
         CW44 : Int;   // Status ID 11: Not Used (0 Hex / 0 Dec)
         CW46 : Int;   // Status ID 12: Not Used (0 Hex / 0 Dec)
      END_STRUCT;
      Tx_I : Struct
         CW18 : Int;   // Status ID 1: Totalizer 1 [kg] (752 Hex / 1874 Dec)
         CW20 : Int;   // Status ID 2: Bin Weigher Fill Weight [kg] (762 Hex / 1890 Dec)
         CW22 : Int;   // Status ID 3: Status 0 + 1 (2D0 Hex / 720 Dec)
         CW24 : Int;   // Status ID 4: Status 8 + 9 (350 Hex / 848 Dec)
         CW26 : Int;   // Status ID 5: Priority Event (610 Hex / 1552 Dec)
         CW28 : Int;   // Status ID 6: Variable ID from faceplate range 1872-2158 (dec)
         CW30 : Int;
      END_STRUCT;
   END_STRUCT;
END_TYPE

TYPE "ACESYS_SIM_PFISTERSDD"
AUTHOR : FLSmidth
FAMILY : ACESYS
NAME : SIM_PFIS
VERSION : 8.0
   STRUCT
      Enable : Bool;
      SSW_Enable : Bool;
      DosingMode : Bool;
      MeasuringMode : Bool;
      FieldMode_Enable : Bool;
      Start : Bool;
      Run_Enable : Bool;
      Run_Const : Bool;
      CorrectionDone : Bool;
      ToggleBit : Bool;
      ToggleBit_Enable : Bool;
      WORK : Struct
         DosingMode : Bool;
         MeasuringMode : Bool;
         FieldMode : Bool;
         Run : Bool;
         CorrectionDone : Bool;
         Togglebit : Bool;
         SSW : Bool;
         Spare0 : Bool;
         Spare1 : Bool;
         Spare2 : Bool;
         Spare3 : Bool;
         Spare4 : Bool;
         Spare5 : Bool;
         Spare6 : Bool;
         Spare7 : Bool;
         Spare8 : Bool;
         SpareInt1 : Int;
         SpareInt2 : Int;
         SpareInt3 : Int;
         SpareReal1 : Real;
         SpareReal2 : Real;
         SpareReal3 : Real;
      END_STRUCT;
   END_STRUCT;
END_TYPE

TYPE "CNT_for_Period"
   STRUCT
      CNT_Begin : Real;
      CNT_Current : Real;
      CNT_Previous : Real;
   END_STRUCT;
END_TYPE

TYPE "ATV9X_CW_IO"
   STRUCT
      pkw_1 : Int;   // PKE
      pkw_2 : Int;   // R/W
      pkw_3 : Int;   // PWE
      pkw_4 : Int;   // PWE
      spare_8 : Bool;
      spare_9 : Bool;
      spare_10 : Bool;
      spare_11 : Bool;
      spare_12 : Bool;
      spare_13 : Bool;
      spare_14 : Bool;
      spare_15 : Bool;
      run_frw : Bool;   // 1 - Run Forward
      run_rvr : Bool;   // 1- Run Revers
      run : Bool;   // 1 - Работа
      spare_3 : Bool;
      spare_4 : Bool;
      spare_5 : Bool;
      spare_6 : Bool;
      rst_flt : Bool;   // Error Reset
      speed_hz_sp : Int;   // 0.1 Hz Reference frequency
      pzd_3 : Int;
      pzd_4 : Int;
      pzd_5 : Int;
      pzd_6 : Int;
      pzd_7 : Int;
      pzd_8 : Int;
      pzd_9 : Int;
      pzd_10 : Int;
      pzd_11 : Int;
      pzd_12 : Int;
      pzd_13 : Int;
      pzd_14 : Int;
      pzd_15 : Int;
      pzd_16 : Int;
   END_STRUCT;
END_TYPE

TYPE "ATV9X_SW_CIA"
   STRUCT
      pkw_1 : Int;   // PKE
      pkw_2 : Int;   // R/W
      pkw_3 : Int;   // PWE
      pkw_4 : Int;   // PWE
      spare_8 : Bool;
      remote : Bool;
      target_reached : Bool;   // Reference value reached
      internal_limit_active : Bool;   // Reference value outside limits
      spare_12 : Bool;
      spare_13 : Bool;
      stop_btn : Bool;   // Manufacturerspecific Stop via STOP key
      revers : Bool;
      rdy_to_sw : Bool;   // 1 = Awaiting power Stage supply
      ready : Bool;   // Ready
      oper_en : Bool;   // Running
      fault : Bool;   // Fault
      v_en : Bool;   // Power stage supply present
      q_stop : Bool;   // 0 = Quick stop is active
      sw_dis : Bool;   // Power stage supply disabled
      warning : Bool;   // A warning is active
      speed_hz : Int;   // 0.1 Hz Motor frequency
      power : Int;   // % Motor power
      power_nominal : Int;   // Nominal motor power
      current : Int;   // Motor current
      speed_hz_max : Int;   // 0.1 Hz
      fault_code : Int;   // Fault code on last fault
      speed_rpm : Int;   // rpm Output velocity
      inputs : Word;   // Logic inputs states
      pzd_10 : Word;   // Logic inputs states
      pzd_11 : Word;
      pzd_12 : Word;
      pzd_13 : Word;
      pzd_14 : Word;
      pzd_15 : Word;
      pzd_16 : Word;
   END_STRUCT;
END_TYPE

TYPE "ATV9X_SW_IO"
   STRUCT
      pkw_1 : Int;   // PKE
      pkw_2 : Int;   // R/W
      pkw_3 : Int;   // PWE
      pkw_4 : Int;   // PWE
      spare_3 : Bool;   // 1: управление по сети; 0: управление через клеммники или графический терминал
      remote : Bool;
      at_speed : Bool;   // 1: задание достигнуто
      ord_out_limits : Bool;   // 1: задание вне ограничений
      spare_4 : Bool;
      spare_5 : Bool;
      stop_btn : Bool;   // 1: остановка осуществлена нажатием клавиши STOP на графическом терминале
      revers : Bool;   // 1: вращение назад
      spare_0 : Bool;   // 0 Зарезервирован (= 0 или 1)
      ready : Bool;   // Готовность ПЧ: 1 -ПЧ готов
      run : Bool;   // 1 - Работа
      fauilt : Bool;   // Состояние обнаруженной ошибки функционирования: 1: активно
      power_on : Bool;   // Силовое питание присутствует: 1 - да
      spare_1 : Bool;
      spare_2 : Bool;
      warning : Bool;   // 1 - Предупреждение
      speed_hz : Int;   // 0.1 Hz Motor frequency
      power : Int;   // % Motor power
      power_nominal : Int;   // Nominal motor power
      current : Int;   // Motor current
      speed_hz_max : Int;   // 0.1 Hz
      fault_code : Int;   // Fault code on last fault
      speed_rpm : Int;   // rpm Output velocity
      inputs : Word;   // Logic inputs states
      pzd_10 : Word;   // Logic inputs states
      pzd_11 : Word;
      pzd_12 : Word;
      pzd_13 : Word;
      pzd_14 : Word;
      pzd_15 : Word;
      pzd_16 : Word;
   END_STRUCT;
END_TYPE

TYPE "ATV9X_CW_CIA"
   STRUCT
      pkw_1 : Int;   // PKE
      pkw_2 : Int;   // R/W
      pkw_3 : Int;   // PWE
      pkw_4 : Int;   // PWE
      Halt : Bool;
      spare_9 : Bool;
      spare_10 : Bool;
      spare_11 : Bool;
      spare_12 : Bool;
      spare_13 : Bool;
      spare_14 : Bool;
      spare_15 : Bool;
      switch_on : Bool;   // Mains contactor control
      enable_voltage : Bool;   // Authorization to supply AC power
      quick_stop : Bool;   // 0 = Quick stop active
      enable_operation : Bool;   // 1 = Run command
      spare_4 : Bool;
      spare_5 : Bool;
      spare_6 : Bool;
      fault_reset : Bool;   // 0 to 1 transition = Error is reset (after cause of error is no longer active)
      speed_hz_sp : Int;   // 0.1 Hz Reference frequency
      pzd_3 : Int;
      pzd_4 : Int;
      pzd_5 : Int;
      pzd_6 : Int;
      pzd_7 : Int;
      pzd_8 : Int;
      pzd_9 : Int;
      pzd_10 : Int;
      pzd_11 : Int;
      pzd_12 : Int;
      pzd_13 : Int;
      pzd_14 : Int;
      pzd_15 : Int;
      pzd_16 : Int;
   END_STRUCT;
END_TYPE

TYPE "ACESYS_MASTER_LINK"
TITLE = ACESYS Master link
AUTHOR : FLSmidth
FAMILY : ACESYS
NAME : Mast_Lnk
VERSION : 8.0
   STRUCT
      Flash_Slow : Bool;   // Slow flash 0.4/0.4 sec
      Flash_Fast : Bool;   // Fast flash 0.2/0.2 sec
      Pulse_Sec : Bool;   // Pulse per Second
      Pulse_Min : Bool;   // Pulse per Minute
      Pulse_Hour : Bool;   // Pulse per Hour
      Pulse_Day : Bool;   // Pulse per Day
      Pulse_Month : Bool;   // Pulse per Month
      Pulse_Year : Bool;   // Pulse per Year
      Sim_Enable : Bool;   // Device Simulation Enabled
      WatchDog_Elap : Bool;   // Watchdog elapsed
      SS_Field_Enable : Bool;   // Single Start from Field
      SS_FP_Enable : Bool;   // Single Start from Faceplate
      Man_Enable : Bool;   // Manual Operation from Faceplate
      Loc_Enable : Bool;   // Local Operation from field
      Test_Enable : Bool;   // Test Operation from faceplate
      LOC_TYPE : Bool;   // "0" = Local operation from PLC / "1" = Local operation from field
      REM_Type : Bool;
      QSTOP_FP_Unit : Bool;
      FIRST_SCAN : Bool;   // First Scan
      SEC_Toggle : Bool;   // Second Toggle
      Spare_02_4 : Bool;
      Spare_02_5 : Bool;
      Spare_02_6 : Bool;
      Spare_02_7 : Bool;
      Spare_03_0 : Bool;
      Spare_03_1 : Bool;
      Spare_03_2 : Bool;
      Spare_03_3 : Bool;
      Spare_03_4 : Bool;
      Spare_03_5 : Bool;
      Spare_03_6 : Bool;
      Spare_03_7 : Bool;
      TimeStamp : Word;   // Time Stamp for HMI
      OB1_CycleTime : Int;
   END_STRUCT;
END_TYPE

TYPE "ACESYS_DEPT_LINK"
TITLE = ACESYS Department link
AUTHOR : FLSmidth
FAMILY : ACESYS
NAME : DEPT_Lnk
VERSION : 8.0
   STRUCT
      TimeStamp : Word;   // Time Stamp for HMI
      OB1_CycleTime : Int;
      Reset : Bool;   // Alarm Reset
      Start : Bool;   // Start
      Stop : Bool;   // Stop
      MasterStop : Bool;   // Master Stop
      QuickStop : Bool;   // Quick Stop
      DeptSelect : Bool;   // Department Select
      DeptDeSelect : Bool;   // Department De-Select
      Flash_Slow : Bool;   // Slow flash 0.4/0.4 sec
      Flash_Fast : Bool;   // Fast flash 0.2/0.2 sec
      FIRST_SCAN : Bool;   // First Scan
      Pulse_1sec : Bool;   // Pulse per Second
      Pulse_1min : Bool;   // Pulse per Minute
      Pulse_1Hour : Bool;   // Pulse per Hour
      Pulse_1Day : Bool;   // Pulse per Day
      Pulse_1Month : Bool;   // Pulse Per month
      Pulse_1Year : Bool;   // Pulse per Year
      Sim_Enable : Bool;   // Device Simulation Enabled
      Man_Enable : Bool;   // Manual operation from faceplate enabled
      Loc_Enable : Bool;   // Local Operation Enabled from field
      Test_Enable : Bool;   // Test Operation enabled
      SS_Field_Enable : Bool;   // Single Start from Field Enabled
      SS_FP_Enable : Bool;   // Single Start from facepalte Enabled
      QSTOP_FP_Unit : Bool;   // Enable Quick Stop from Unit Faceplate
      EmergencyStop : Bool;   // Department Emergency Stop
      All_Group_ON : Bool;   // All Groups On
      All_Group_OFF : Bool;   // All Groups Off
      All_Group_Sel_RDY : Bool;   // All Groups Selected is Ready
      All_Selected : Bool;   // All Groups Selected
      All_DeSelected : Bool;   // All Groups De-selected
      All_Selected_Running : Bool;   // All Selected groups is running
      Ready_For_StopCmd : Bool;   // Some Groups De-selcted, but running
      WatchDog_Failure : Bool;   // Watchdog Communication Failure with HMI
      LOC_TYPE : Bool;   // "0" = Local operation from PLC / "1" = Local operation from field
      REM_Type : Bool;   // "1" Force to Local Mode
      SEC_Toggle : Bool;   // Second Toggle
      SpareBool_13 : Bool;
      SpareBool_12 : Bool;
      SpareBool_11 : Bool;
      SpareBool_10 : Bool;
      SpareBool_09 : Bool;
      SpareBool_08 : Bool;
      SpareBool_07 : Bool;
      SpareBool_06 : Bool;
      SpareBool_05 : Bool;
      SpareBool_04 : Bool;
      SpareBool_03 : Bool;
      SpareBool_02 : Bool;
      SpareBool_01 : Bool;
   END_STRUCT;
END_TYPE

TYPE "ACESYS_TOKEN"
TITLE = ACESYS Token
AUTHOR : FLSmidth
FAMILY : ACESYS
NAME : TOKEN
VERSION : 8.0
   STRUCT
      TimeStamp : Word;   // Timestamp for reporting to ECS
      OB1_CycleTime : Int;
      Acknowledge : Bool;
      AL_UNIT : Bool;   // Unit Alarm OK
      StartWarn : Bool;   // Start Warning
      GON : Bool;   // Group on
      GOFF : Bool;   // Group off
      Interlock_Unit : Bool;
      DeSelButRun : Bool;   // A Unit or Route is De-selected, but still running
      Sim_Enable : Bool;   // Device Simulation Enabled
      Flash_Slow : Bool;   // Flash slow for lamp inidcation
      Flash_Fast : Bool;   // Flash fast for lamp inidcation
      Pulse_1sec : Bool;   // 1 Seconds Puls
      Pulse_1min : Bool;   // 1 Minute Puls
      Pulse_1Hour : Bool;
      Pulse_1Day : Bool;
      Pulse_1Month : Bool;
      Pulse_1Year : Bool;
      EmergencyStop : Bool;   // Emergency stop ("1" = Ok)
      ModeSwap : Bool;
      SS_Field_Enable : Bool;
      SS_FP_Enable : Bool;
      Man_Enable : Bool;   // Enable Manual operation from faceplate
      Loc_Enable : Bool;   // Enable Local operation from field
      TEST_Enable : Bool;   // Enable Test operation from faceplate
      LOC_TYPE : Bool;   // "0" = Local operation from PLC / "1" = Local operation from field
      REM_TYPE : Bool;
      QSTOP_FP_Unit : Bool;
      AllUnitsAuto : Bool;
      NotEmpty : Bool;
      CheckNotEmpty : Bool;
      ResetNotEmpty : Bool;
      AlarmSuppres : Bool;
      SACK_On : Bool;
      SACK_Off : Bool;
      FIRST_SCAN : Bool;   // First Scan
      SEC_Toggle : Bool;   // Second Toggle
      UnitSelect : Bool;   // If '0' no units in group have the SEL input set
      SpareBool_12 : Bool;
      SpareBool_11 : Bool;
      SpareBool_10 : Bool;
      SpareBool_09 : Bool;
      SpareBool_08 : Bool;
      SpareBool_07 : Bool;
      SpareBool_06 : Bool;
      SpareBool_05 : Bool;
      SpareBool_04 : Bool;
      SpareBool_03 : Bool;
      SpareBool_02 : Bool;
      SpareBool_01 : Bool;
   END_STRUCT;
END_TYPE

TYPE "ACESYS_GRP_CMD"
TITLE = ACESYS Department Commands
AUTHOR : FLSmidth
FAMILY : ACESYS
NAME : GRP_CMD
VERSION : 8.0
   STRUCT
      GSEL : Bool;   // Group Select
      GSTR : Bool;   // Group Start
      GSTP : Bool;   // Group Stop
      GQSTP : Bool;   // Group Quick Stop
      GSS_FP : Bool;   // Group Single Start from Faceplate
      GSS_Field : Bool;   // Group Single Start from Field
      GLTP : Bool;   // Group Local Test Permission
      GASTW : Bool;   // Group Audible Start
   END_STRUCT;
END_TYPE

TYPE "ACESYS_INTL"
TITLE = ACESYS Interlock Data
AUTHOR : FLSmidth
FAMILY : ACESYS
NAME : INTL
VERSION : 8.0
   STRUCT
      OK : Bool;   // Bit 0: Interlock fulfilled
      DetectFirst : Bool;   // Bit 1: Detect first occuring interlock, unit running
      Bit2 : Bool;
      ClearFirst : Bool;   // Bit 3: Clear first Interlock
      Bit4 : Bool;
      Bit5 : Bool;
      Bit6 : Bool;
      Bit7 : Bool;
   END_STRUCT;
END_TYPE

TYPE "ACESYS_HLC_LINK"
TITLE = ACESYS HLC Link
AUTHOR : FLSmidth
FAMILY : ACESYS
NAME : HLC_Lnk
VERSION : 8.0
   STRUCT
      GR01_Enable : Bool;   // Enable High Level Control for Group 01
      GR02_Enable : Bool;   // Enable High Level Control for Group 02
      GR03_Enable : Bool;   // Enable High Level Control for Group 03
      GR04_Enable : Bool;   // Enable High Level Control for Group 04
      GR05_Enable : Bool;   // Enable High Level Control for Group 05
      GR06_Enable : Bool;   // Enable High Level Control for Group 06
      GR07_Enable : Bool;   // Enable High Level Control for Group 07
      GR08_Enable : Bool;   // Enable High Level Control for Group 08
      GR09_Enable : Bool;   // Enable High Level Control for Group 09
      GR10_Enable : Bool;   // Enable High Level Control for Group 10
      Spare_01 : Bool;   // Spare
      Spare_02 : Bool;   // Spare
      Spare_03 : Bool;   // Spare
      Spare_04 : Bool;   // Spare
      Spare_05 : Bool;   // Spare
      Spare_06 : Bool;   // Spare
   END_STRUCT;
END_TYPE

TYPE "ACESYS_HMI_STAT_32T"
TITLE = ACESYS Status to HMI - 32 bit MSW + Timestamp
AUTHOR : FLSmidth
FAMILY : ACESYS
NAME : STAT_32T
VERSION : 8.0
   STRUCT
      EXT : Struct
         AlarmWarnUnAck : Bool;   // Bit 24: Alarm Warning Present or Unacknowledged
         AckRequired : Bool;   // Bit 25: Acknowledge Required
         Maintanence : Bool;   // Bit 26: Maintanence
         Operation : Bool;   // Bit 27: In Operation
         Forced : Bool;   // Bit 28: Forced
         BIT29 : Bool;   // Bit 29
         BIT30 : Bool;   // Bit 30
         BIT31 : Bool;   // Bit 31
         ModeBit1 : Bool;   // Bit 16: Mode bit 1 (value = 1)
         ModeBit2 : Bool;   // Bit 17: Mode bit 2 (value = 2)
         ModeBit3 : Bool;   // Bit 18: Mode bit 3 (value = 4)
         BIT19 : Bool;   // Bit 19
         BIT20 : Bool;   // Bit 20
         AlarmSuppressed : Bool;   // Bit 21: Alarm Suppressed
         AlarmPresent : Bool;   // Bit 22: Alarm Condition Present
         AlarmFailUnAck : Bool;   // Bit 23: Alarm Failure Present or Unacknowledged
      END_STRUCT;
      Status : Int;
      TimeStamp : Word;
   END_STRUCT;
END_TYPE

TYPE "ACESYS_HMI_STAT_16T"
TITLE = ACESYS Status to HMI - 16 bit MSW + Timestamp
AUTHOR : FLSmidth
FAMILY : ACESYS
NAME : STAT_16T
VERSION : 8.0
   STRUCT
      Status : Int;
      TimeStamp : Word;
   END_STRUCT;
END_TYPE

TYPE "ACESYS_HMI_STAT_ANALOG"
TITLE = ACESYS Status to HMI - Value + Trig Val +32 bit MSW + Timestamp
AUTHOR : FLSmidth
FAMILY : ACESYS
NAME : ANALOG
VERSION : 8.0
   STRUCT
      VALUE : Real;   // Analog Value
      TRIGVALUE : Real;   // Alarm Trig Value
      EXT : Struct
         AlarmWarnUnAck : Bool;   // Bit 24: Alarm Warning Present or Unacknowledged
         AckRequired : Bool;   // Bit 25: Acknowledge Required
         Maintanence : Bool;   // Bit 26: Maintanence
         Operation : Bool;   // Bit 27: In Operation
         Forced : Bool;   // Bit 28: Forced
         BIT29 : Bool;   // Bit 29
         BIT30 : Bool;   // Bit 30
         BIT31 : Bool;   // Bit 31
         ModeBit1 : Bool;   // Bit 16: Mode bit 1 (value = 1)
         ModeBit2 : Bool;   // Bit 17: Mode bit 2 (value = 2)
         ModeBit3 : Bool;   // Bit 18: Mode bit 3 (value = 4)
         BIT19 : Bool;   // Bit 19
         BIT20 : Bool;   // Bit 20
         AlarmSuppressed : Bool;   // Bit 21: Alarm Suppressed
         AlarmPrsent : Bool;   // Bit 22: Alarm Condition Present
         AlarmFailUnAck : Bool;   // Bit 23: Alarm Failure Present or Unacknowledged
      END_STRUCT;
      Status : Int;
      TimeStamp : Word;
   END_STRUCT;
END_TYPE

TYPE "ACESYS_HMI_STAT_16"
TITLE = ACESYS Status to HMI - 16 bit MSW
AUTHOR : FLSmidth
FAMILY : ACESYS
NAME : STAT_16
VERSION : 8.0
   STRUCT
      Status : Int;
   END_STRUCT;
END_TYPE

TYPE "ACESYS_ADPT_MOTOR"
TITLE = Data Structure for Adaptor block (data exchange with HMI)
AUTHOR : FLSmidth
FAMILY : ACESYS
NAME : ADPT
VERSION : 8.0
   STRUCT
      Intell_Type : Int;
      VersionNo : Int;
      BuildNo : Int;
      FuncType : Int;
      Options : Int;
      NetNo : Int;
      NodeNo : Int;
      Sim_Enable : Bool;   // Device Simulation Enabled
      Flash_Slow : Bool;   // Flash slow for lamp inidcation
      Flash_Fast : Bool;   // Flash fast for lamp inidcation
      Pulse_1sec : Bool;   // 1 Seconds Puls
      CON1 : Bool;
      CON2 : Bool;
      CON3 : Bool;
      RES : Bool;
      LOC : Bool;
      MAN : Bool;
      SS : Bool;
      TESTP : Bool;
      Indication : Bool;   // Type Indication
      SpareBool03 : Bool;
      SpareBool02 : Bool;
      SpareBool01 : Bool;
      HMI_INT : Array[1..70] of Int;
      HMI_REAL : Array[1..16] of Real;
      HMI_BOOL : Array[1..160] of Bool;
   END_STRUCT;
END_TYPE

TYPE "ACESYS_BQ16"
TITLE = Data Structure for exchange data between BQ16_Ctrl / BQ16_prgm
AUTHOR : FLSmidth
FAMILY : ACESYS
NAME : AirBlast
VERSION : 8.0
   STRUCT
      SEL : Bool;   // Select
      Start : Bool;   // Start
      Reset : Bool;   // Reset Program Sequence
      BQ_CMD : Array[0..16] of Bool;   // Blast Commands
      SelectProgram : Int;   // Selected program
      ProgramIncrement : Int;   // Count Number of programs (+1/prg. routine)
      NumberBlasters : Int := 16;   // Number of Blasters to be Used
      Spare_Int_01 : Int := 16;
   END_STRUCT;
END_TYPE

TYPE "ACESYS_PlcToPLC"
TITLE = PLC to PLC Communication Data Layout
AUTHOR : FLSmidth
FAMILY : ACESYS
NAME : PLCtoPLC
VERSION : 8.0
   STRUCT
      Watchdog : Bool;   // Watchdog Bit
      Simulation_Enabled : Bool;   // Device Simulation Enabled
      Spare_2 : Bool;   // Not Used
      Spare_3 : Bool;   // Not Used
      Spare_4 : Bool;   // Not Used
      Spare_5 : Bool;   // Not Used
      Spare_6 : Bool;   // Not Used
      Spare_7 : Bool;   // Not Used
      BOOLEAN : Array[0..63] of Bool;   // Boolean Data
      REAL_VAL : Array[0..15] of Real;   // Real Data
      INT_VAL : Array[0..15] of Int;   // Interger Data
   END_STRUCT;
END_TYPE

TYPE "ACESYS_PowerLink"
TITLE = Data Structure for Adapter block for POWER block
AUTHOR : FLSmidth
FAMILY : ACESYS
NAME : PWR_Lnk
VERSION : 8.0
   STRUCT
      INFO : Struct
         BlockFunction : Int;   // 0 = Power Monitor, 1 = MV Feeder, 2 = MV Motor
         Intell_Type : Int;   // Intelligent Device Type
         BuildNo : Int;   // Adaptor Block Build Number
         ADAPT_FuncType : Int;   // Feeder Type
         ADAPT_Option : Int;   // For Future Use from ADAPT
         NetNo : Int;   // Device Net Number
         NodeNo : Int;   // Device Node Number
         Sim_Enable : Bool;   // Device Simulation Enabled
         Flash_Slow : Bool;   // Flash slow for lamp inidcation
         Flash_Fast : Bool;   // Flash fast for lamp inidcation
         Pulse_1sec : Bool;   // 1 Seconds Puls
         Pulse_1min : Bool;   // 1 Minute Puls
         Pulse_1Hour : Bool;   // 1 Hour Puls
         Pulse_1Day : Bool;   // 1 Day Puls
         Pulse_1Month : Bool;   // 1 Month Puls
         Pulse_1Year : Bool;   // 1 Year Puls
         FIRST_SCAN : Bool;   // First Scan
         SEC_Toggle : Bool;   // Second Toggle
         Spare05 : Bool;   // Spare
         Spare04 : Bool;   // Spare
         Spare03 : Bool;   // Spare
         Spare02 : Bool;   // Spare
         Spare01 : Bool;   // Spare
      END_STRUCT;
      SEL : Struct   // Enginering range to be used in faceplate
         A_kA : Bool;   // A or kA
         V_kV : Bool;   // V or kV
         kW_MW : Bool;   // kW or MW
         kWh_MWh : Bool;   // kWh or MWh
         C_F : Bool;   // Celsius or Farenheit
         Spare01 : Bool;
         Spare02 : Bool;
         Spare03 : Bool;
         Spare04 : Bool;
         Spare05 : Bool;
         Spare06 : Bool;
         Spare07 : Bool;
         Spare08 : Bool;
         Spare09 : Bool;
         Spare10 : Bool;
         Spare11 : Bool;
      END_STRUCT;
      Status : Struct   // Electric Power System Device Fucntion Status
         BUSF : Bool;   // Communication Healthy
         HLTY : Bool;   // Device Healthy
         ACK : Bool;   // Acknowledge Received
         Spare13 : Bool;   // Spare
         Spare12 : Bool;   // Spare
         Spare11 : Bool;   // Spare
         Spare10 : Bool;   // Spare
         Spare09 : Bool;   // Spare
         Spare08 : Bool;   // Spare
         Spare07 : Bool;   // Spare
         Spare06 : Bool;   // Spare
         Spare05 : Bool;   // Spare
         Spare04 : Bool;   // Spare
         Spare03 : Bool;   // Spare
         Spare02 : Bool;   // Spare
         Spare01 : Bool;   // Spare
      END_STRUCT;
      Command : Struct
         RES : Bool;   // Reset Command
         Spare15 : Bool;
         Spare14 : Bool;
         Spare13 : Bool;
         Spare12 : Bool;
         Spare11 : Bool;
         Spare10 : Bool;
         Spare09 : Bool;
         Spare08 : Bool;
         Spare07 : Bool;
         Spare06 : Bool;
         Spare05 : Bool;
         Spare04 : Bool;
         Spare03 : Bool;
         Spare02 : Bool;
         Spare01 : Bool;   // Reset
      END_STRUCT;
      EN : Struct   // Signals Enabled
         VOLT_LNPH : Bool;   // Phase to pahse & Line to Neutral Voltage V/kV)
         CURR_LN : Bool;   // Line Current
         APOW_PH : Bool;   // Phase Power kW/MW)
         FRQ : Bool;   // Frequency (Hz)
         APOW_AVG : Bool;   // Average Apparent Power (kVA/MVA)
         RTPOW_AVG : Bool;   // Average Reactive Power (kW/MW)
         VOLT_UNBAL : Bool;   // Voltage Unbalance (%)
         CURR_UNBAL : Bool;   // Current unbalance (%)
         VOLT_THD : Bool;   // Total Hormonic Distorsion Voltage (%)
         CURR_THD : Bool;   // Total Hormonic Distorsion Current (%)
         RENG : Bool;   // Average Reactive Energy (kVARH/MVARH)
         kWH_REV : Bool;   // Reverse kWH (kWhr/MWhr)
         kVAH_FwdRev : Bool;   // kVAH Forward/Reverse(kVAH/MVAH)
         kVARH_Rev : Bool;   // kVARH Reverse(kVARH/MVARH)
         MD_kW_Fwd : Bool;   // kW Forward (kW/MW)
         MD_kW_Rev : Bool;   // kW Reverse (kW/MW)
         MD_kVAr_Fwd : Bool;   // kVA Forward (kVAr/MVAr)
         MD_kVAr_Rev : Bool;   // kVA Reverse (kVAr/MVAr)
         HORM_5TH : Bool;   // 5th Order Hormonics
         HORM_7TH : Bool;   // 7th Order Hormonics
         HORM_11TH : Bool;   // 11th Order Hormonics
         MWT : Bool;   // Motor Winding temperature
         MBT : Bool;   // Motor Bearing temperature
         TWT : Bool;   // Transformer Winding temperature
         TOT : Bool;   // Transformer Oil temperature
         RunHrs : Bool;   // Run Hours
         PB_Reset : Bool;   // Enable Reset
         Spare21 : Bool;
         Spare20 : Bool;
         Spare19 : Bool;
         Spare18 : Bool;
         Spare17 : Bool;
         Spare16 : Bool;
         Spare15 : Bool;
         Spare14 : Bool;
         Spare13 : Bool;
         Spare12 : Bool;
         Spare11 : Bool;
         Spare10 : Bool;
         Spare09 : Bool;
         Spare08 : Bool;
         Spare07 : Bool;
         Spare06 : Bool;
         Spare05 : Bool;
         Spare04 : Bool;
         Spare03 : Bool;
         Spare02 : Bool;
         Spare01 : Bool;
      END_STRUCT;
      PARM : Struct
         VOLT_L1L2 : Real;   // L1 Phase to L2 pahse Voltage(V/kV)
         VOLT_L2L3 : Real;   // L2 Phase to L3 pahse Voltage(V/kV)
         VOLT_L3L1 : Real;   // L3 Phase to L1 pahse Voltage(V/kV)
         VOLT_AVG : Real;   // Line to Line Voltage - Average (V/kV)
         CURR_L1 : Real;   // Line Current L1 Phase (A/kA)
         CURR_L2 : Real;   // Line Current L2 Phase (A/kA)
         CURR_L3 : Real;   // Line Current L3 Phase (A/kA)
         CURR_AVG : Real;   // Average Current (A/kA)
         APOW_L1 : Real;   // L1 Phase Power (kW/MW)
         APOW_L2 : Real;   // L2 Phase Power (kW/MW)
         APOW_L3 : Real;   // L3 Phase Power (kW/MW)
         FRQ : Real;   // Frequency (Hz)
         PF_AVG : Real;   // Average Power Factor
         APOW_AVG : Real;   // Average Apparent Power (kVA/MVA)
         RLPOW_AVG : Real;   // Average Real Power (kW/MW)
         RTPOW_AVG : Real;   // Average Reactive Power (kW/MW)
         VOLT_UNBAL : Real;   // Voltage Unbalance (%)
         CURR_UNBAL : Real;   // Current unbalance (%)
         VOLT_THD : Real;   // Total Hormonic Distorsion Voltage (%)
         CURR_THD : Real;   // Total Hormonic Distorsion Current (%)
         AENG : Real;   // Average Active Energy [Forward] (kWhr/MWhr)
         RENG : Real;   // Average Reactive Energy [Forward] (kVARH/MVARH)
         kWH_REV : Real;   // Reverse kWH (kWhr/MWhr)
         kVAH_FwdRev : Real;   // kVAH Forward/Reverse(kVAH/MVAH)
         kVARH_Rev : Real;   // kVARH Reverse(kVARH/MVARH)
         MD_kW_Fwd : Real;   // kW Forward (kW/MW)
         MD_kW_Rev : Real;   // kW Reverse (kW/MW)
         MD_kVAr_Fwd : Real;   // kVA Forward (kVAr/MVA)
         MD_kVAr_Rev : Real;   // kVA Reverse (kVAr/MVA)
         HORM_5TH : Real;   // 5th Order Hormonics
         HORM_7TH : Real;   // 7th Order Hormonics
         HORM_11TH : Real;   // 11th Order Hormonics
         MWT : Real;   // Motor Winding Temperature
         MBT : Real;   // Motor Bearing Temperature
         TWT : Real;   // Transformer Winding temperature
         TOT : Real;   // Transformer Oil temperature
         RunHrs : Real;   // Run Hours
         AI_Spare01 : Real;
         AI_Spare02 : Real;
         AI_Spare03 : Real;
      END_STRUCT;
   END_STRUCT;
END_TYPE

TYPE "ACESYS_PlcToPLC_434Byte"
TITLE = PLC to PLC Communication Data Layout
AUTHOR : FLSmidth
FAMILY : ACESYS
NAME : PLCtoPLC
VERSION : 8.0
   STRUCT
      Watchdog : Bool;   // Watchdog Bit
      Simulation_Enabled : Bool;   // Device Simulation Enabled
      Spare_2 : Bool;   // Not Used
      Spare_3 : Bool;   // Not Used
      Spare_4 : Bool;   // Not Used
      Spare_5 : Bool;   // Not Used
      Spare_6 : Bool;   // Not Used
      Spare_7 : Bool;   // Not Used
      BOOLEAN : Array[0..127] of Bool;   // Boolean Data
      REAL_VAL : Array[0..95] of Real;   // Real Data
      INT_VAL : Array[0..15] of Int;   // Interger Data
   END_STRUCT;
END_TYPE

TYPE "ACESYS_SIM_ALARM"
TITLE = Device Simulation Data for Alarm
AUTHOR : FLSmidth
FAMILY : ACESYS
NAME : SIM_ALM
VERSION : 8.0
   STRUCT
      Enable : Bool;
      SIG_Enable : Bool := TRUE;
      PWR_Enable : Bool := TRUE;
      Spare04 : Bool;
      Spare05 : Bool;
      Spare06 : Bool;
      Spare07 : Bool;
      Spare08 : Bool;
      Spare09 : Bool;
      Spare10 : Bool;
      Spare11 : Bool;
      Spare12 : Bool;
      Spare13 : Bool;
      Spare14 : Bool;
      Spare15 : Bool;
   END_STRUCT;
END_TYPE

